Yaskawa INFORM job: u_tourne2TRJ4.JBI

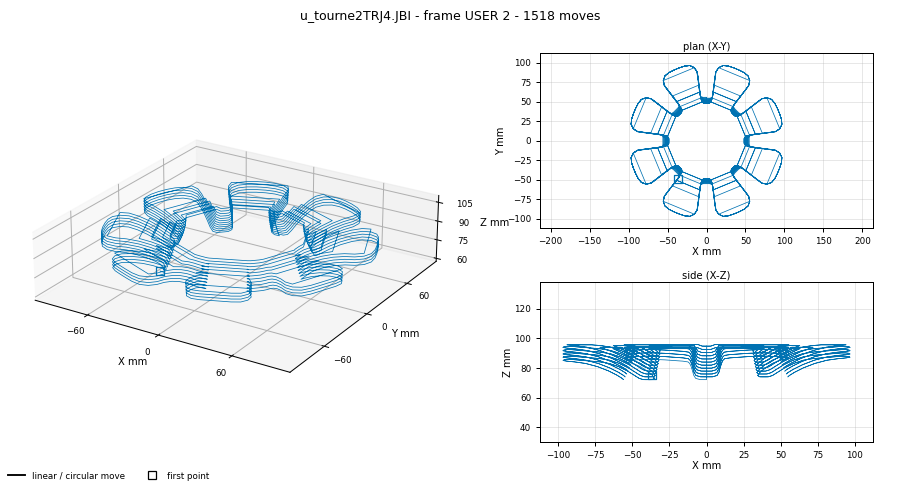
[picture p0: tool path of u_tourne2TRJ4.JBI in frame USER 2, 1518 of 1518 moves have a stored position in this frame; points joined in program order, loops and branches not executed]
/JOB
//NAME u_tourne2TRJ4
///FOLDERNAME DEMO
//POS
///NPOS 1518,0,0,0,0,0
///USER 2
///TOOL 7
///POSTYPE USER
///RECTAN
///RCONF 1,0,0,0,0,0,0,0,0,0,0,0,0,0,0,0,0,0,0,0,0,0,0,0
C00000=-36.517,-48.718,75.143,178.8248,-1.7081,0.0000
C00001=-35.037,-45.351,73.015,-179.8799,17.3496,0.0000
C00002=-36.538,-42.505,72.166,160.0584,24.5518,0.0000
C00003=-38.303,-40.803,72.129,156.0394,22.3811,0.0000
C00004=-39.567,-39.567,72.154,156.8184,23.1816,0.0000
C00005=-40.803,-38.303,72.129,157.6189,23.9606,0.0000
C00006=-42.506,-36.538,72.166,155.4482,19.9416,0.0000
C00007=-45.352,-35.037,73.015,162.6504,-0.1201,0.0000
C00008=-48.718,-36.517,75.143,-178.2919,1.1752,0.0000
C00009=-53.324,-40.007,78.036,-176.9022,2.2727,0.0000
C00010=-59.196,-44.618,80.927,-176.4763,2.6299,0.0000
C00011=-65.578,-49.604,83.062,-176.2458,2.8088,0.0000
C00012=-71.524,-53.949,84.088,-176.0063,2.0395,0.0000
C00013=-77.795,-55.184,84.621,-177.1914,-0.2581,0.0000
C00014=-83.601,-53.037,85.050,-178.9055,-0.7851,0.0000
C00015=-87.741,-47.957,85.481,-179.9599,-0.0745,0.0000
C00016=-90.934,-41.602,85.762,-179.9943,-0.0115,0.0000
C00017=-93.717,-34.883,85.762,-179.9943,-0.0115,0.0000
C00018=-95.953,-28.131,85.481,-179.9771,-0.0859,0.0000
C00019=-96.617,-21.612,85.050,179.7822,-1.3294,0.0000
C00020=-94.030,-15.989,84.621,178.1936,-2.1673,0.0000
C00021=-88.723,-12.427,84.088,175.7376,-1.3849,0.0000
C00022=-81.446,-11.295,83.062,175.3653,-0.6668,0.0000
C00023=-73.408,-10.308,80.927,175.6470,-0.6321,0.0000
C00024=-65.995,-9.417,78.036,176.2042,-0.5857,0.0000
C00025=-60.270,-8.627,75.143,177.9597,-0.3784,0.0000
C00026=-56.844,-7.293,73.015,-167.4661,12.3794,0.0000
C00027=-55.892,-4.219,72.166,-176.1983,30.0937,0.0000
C00028=-55.936,-1.768,72.129,178.6805,31.1908,0.0000
C00029=-55.957,0.000,72.154,180.0000,31.1976,0.0000
C00030=-55.936,1.767,72.129,-178.6805,31.1908,0.0000
C00031=-55.892,4.220,72.166,176.1916,30.0937,0.0000
C00032=-56.844,7.293,73.015,167.4661,12.3794,0.0000
C00033=-60.270,8.627,75.143,-177.9597,-0.3784,0.0000
C00034=-65.995,9.417,78.036,-176.2042,-0.5857,0.0000
C00035=-73.408,10.308,80.927,-175.6470,-0.6321,0.0000
C00036=-81.446,11.295,83.062,-175.3653,-0.6668,0.0000
C00037=-88.723,12.427,84.088,-175.7376,-1.3849,0.0000
C00038=-94.030,15.989,84.621,-178.1936,-2.1673,0.0000
C00039=-96.617,21.612,85.050,-179.7822,-1.3294,0.0000
C00040=-95.953,28.131,85.481,179.9771,-0.0859,0.0000
C00041=-93.717,34.883,85.762,179.9943,-0.0115,0.0000
C00042=-90.934,41.602,85.762,179.9943,-0.0115,0.0000
C00043=-87.741,47.957,85.481,179.9599,-0.0745,0.0000
C00044=-83.601,53.037,85.050,178.9055,-0.7851,0.0000
C00045=-77.795,55.184,84.621,177.1914,-0.2581,0.0000
C00046=-71.524,53.949,84.088,176.0063,2.0395,0.0000
C00047=-65.578,49.604,83.062,176.2458,2.8088,0.0000
C00048=-59.196,44.618,80.927,176.4763,2.6299,0.0000
C00049=-53.324,40.007,78.036,176.9022,2.2727,0.0000
C00050=-48.718,36.517,75.143,178.2919,1.1752,0.0000
C00051=-45.351,35.037,73.015,-162.6504,-0.1201,0.0000
C00052=-42.505,36.538,72.166,-155.4482,19.9416,0.0000
C00053=-40.803,38.303,72.129,-157.6189,23.9606,0.0000
C00054=-39.567,39.567,72.154,-156.8184,23.1816,0.0000
C00055=-38.303,40.803,72.129,-156.0394,22.3811,0.0000
C00056=-36.538,42.506,72.166,-160.0584,24.5518,0.0000
C00057=-35.037,45.352,73.015,179.8799,17.3496,0.0000
C00058=-36.517,48.718,75.143,-178.8248,-1.7081,0.0000
C00059=-40.007,53.324,78.036,-177.7273,-3.0978,0.0000
C00060=-44.618,59.196,80.927,-177.3701,-3.5237,0.0000
C00061=-49.604,65.578,83.062,-177.1912,-3.7542,0.0000
C00062=-53.949,71.524,84.088,-177.9605,-3.9937,0.0000
C00063=-55.184,77.795,84.621,179.7419,-2.8086,0.0000
C00064=-53.037,83.601,85.050,179.2149,-1.0945,0.0000
C00065=-47.957,87.741,85.481,179.9255,-0.0401,0.0000
C00066=-41.602,90.934,85.762,179.9885,-0.0057,0.0000
C00067=-34.883,93.717,85.762,179.9885,-0.0057,0.0000
C00068=-28.131,95.953,85.481,179.9141,-0.0229,0.0000
C00069=-21.612,96.617,85.050,178.6706,0.2178,0.0000
C00070=-15.989,94.030,84.621,177.8327,1.8064,0.0000
C00071=-12.427,88.723,84.088,178.6151,4.2624,0.0000
C00072=-11.295,81.446,83.062,179.3332,4.6347,0.0000
C00073=-10.308,73.408,80.927,179.3679,4.3530,0.0000
C00074=-9.417,65.995,78.036,179.4143,3.7958,0.0000
C00075=-8.627,60.270,75.143,179.6216,2.0403,0.0000
C00076=-7.293,56.844,73.015,-167.6206,-12.5339,0.0000
C00077=-4.220,55.892,72.166,-149.9063,-3.8084,0.0000
C00078=-1.767,55.936,72.129,-148.8092,1.3195,0.0000
C00079=0.000,55.957,72.154,-148.8024,-0.0000,0.0000
C00080=0.000,54.840,74.049,-150.2587,-0.0000,0.0000
C00081=1.666,54.823,74.024,-150.2658,-1.1877,0.0000
C00082=4.048,54.790,74.062,-151.4221,3.8700,0.0000
C00083=7.088,55.804,74.943,-168.9171,11.6612,0.0000
C00084=8.393,59.388,77.145,179.6273,-2.1319,0.0000
C00085=9.180,65.335,80.122,179.4719,-3.5317,0.0000
C00086=10.089,72.980,83.074,179.4487,-3.8705,0.0000
C00087=11.094,81.206,85.240,179.4429,-3.9856,0.0000
C00088=12.226,88.613,86.276,178.8517,-3.5956,0.0000
C00089=15.808,94.009,86.813,178.2001,-1.5192,0.0000
C00090=21.475,96.642,87.246,178.8998,-0.1834,0.0000
C00091=28.048,95.980,87.679,179.9312,0.0229,0.0000
C00092=34.856,93.728,87.962,179.9943,0.0057,0.0000
C00093=41.629,90.922,87.962,179.9943,0.0057,0.0000
C00094=48.035,87.701,87.679,179.9370,0.0344,0.0000
C00095=53.151,83.521,87.246,179.3525,0.9054,0.0000
C00096=55.296,77.652,86.813,179.7993,2.3440,0.0000
C00097=54.014,71.304,86.276,-178.2664,3.3554,0.0000
C00098=49.577,65.266,85.240,-177.5775,3.2132,0.0000
C00099=44.470,58.738,83.074,-177.6468,3.1267,0.0000
C00100=39.708,52.690,80.122,-177.8713,2.8736,0.0000
C00101=36.059,47.928,77.145,-178.7560,1.7711,0.0000
C00102=34.447,44.472,74.943,179.5711,-15.8793,0.0000
C00103=35.880,41.605,74.062,-161.3594,-23.4144,0.0000
C00104=37.588,39.944,74.024,-157.2874,-21.2658,0.0000
C00105=38.778,38.778,74.049,-158.0009,-21.9991,0.0000
C00106=39.943,37.588,74.024,-158.7342,-22.7126,0.0000
C00107=41.605,35.880,74.062,-156.5880,-18.6327,0.0000
C00108=44.472,34.447,74.943,-164.1207,0.4289,0.0000
C00109=47.928,36.059,77.145,178.2289,-1.2440,0.0000
C00110=52.690,39.708,80.122,177.1264,-2.1287,0.0000
C00111=58.738,44.470,83.074,176.8733,-2.3532,0.0000
C00112=65.266,49.577,85.240,176.7868,-2.4225,0.0000
C00113=71.304,54.014,86.276,176.6446,-1.7336,0.0000
C00114=77.652,55.296,86.813,177.6560,0.2007,0.0000
C00115=83.521,53.151,87.246,179.0946,0.6475,0.0000
C00116=87.701,48.035,87.679,179.9656,0.0630,0.0000
C00117=90.922,41.629,87.962,179.9943,0.0057,0.0000
C00118=93.728,34.856,87.962,179.9943,0.0057,0.0000
C00119=95.980,28.048,87.679,179.9771,0.0688,0.0000
C00120=96.642,21.475,87.246,-179.8166,1.1002,0.0000
C00121=94.009,15.808,86.813,-178.4808,1.7999,0.0000
C00122=88.613,12.226,86.276,-176.4044,1.1483,0.0000
C00123=81.206,11.094,85.240,-176.0144,0.5571,0.0000
C00124=72.980,10.089,83.074,-176.1295,0.5513,0.0000
C00125=65.335,9.180,80.122,-176.4683,0.5281,0.0000
C00126=59.388,8.393,77.145,-177.8681,0.3727,0.0000
C00127=55.804,7.088,74.943,168.3388,-11.0829,0.0000
C00128=54.790,4.048,74.062,176.1300,-28.5779,0.0000
C00129=54.823,1.666,74.024,-178.8123,-29.7342,0.0000
C00130=54.840,0.000,74.049,-180.0000,-29.7413,0.0000
C00131=54.823,-1.665,74.024,178.8123,-29.7342,0.0000
C00132=54.790,-4.048,74.062,-176.1304,-28.5752,0.0000
C00133=55.804,-7.088,74.943,-168.3388,-11.0829,0.0000
C00134=59.388,-8.393,77.145,177.8681,0.3727,0.0000
C00135=65.335,-9.180,80.122,176.4683,0.5281,0.0000
C00136=72.980,-10.089,83.074,176.1295,0.5513,0.0000
C00137=81.206,-11.094,85.240,176.0144,0.5571,0.0000
C00138=88.613,-12.226,86.276,176.4044,1.1483,0.0000
C00139=94.009,-15.808,86.813,178.4808,1.7999,0.0000
C00140=96.642,-21.475,87.246,179.8166,1.1002,0.0000
C00141=95.980,-28.048,87.679,-179.9771,0.0688,0.0000
C00142=93.728,-34.856,87.962,-179.9943,0.0057,0.0000
C00143=90.922,-41.629,87.962,-179.9943,0.0057,0.0000
C00144=87.701,-48.035,87.679,-179.9656,0.0630,0.0000
C00145=83.521,-53.151,87.246,-179.0946,0.6475,0.0000
C00146=77.652,-55.296,86.813,-177.6560,0.2007,0.0000
C00147=71.304,-54.014,86.276,-176.6446,-1.7336,0.0000
C00148=65.266,-49.577,85.240,-176.7868,-2.4225,0.0000
C00149=58.738,-44.470,83.074,-176.8733,-2.3532,0.0000
C00150=52.690,-39.708,80.122,-177.1264,-2.1287,0.0000
C00151=47.928,-36.059,77.145,-178.2289,-1.2440,0.0000
C00152=44.472,-34.447,74.943,164.1207,0.4289,0.0000
C00153=41.605,-35.880,74.062,156.5856,-18.6406,0.0000
C00154=39.944,-37.588,74.024,158.7342,-22.7126,0.0000
C00155=38.778,-38.778,74.049,158.0009,-21.9991,0.0000
C00156=37.588,-39.943,74.024,157.2874,-21.2658,0.0000
C00157=35.880,-41.605,74.062,161.3673,-23.4120,0.0000
C00158=34.447,-44.472,74.943,-179.5711,-15.8793,0.0000
C00159=36.059,-47.928,77.145,178.7560,1.7711,0.0000
C00160=39.708,-52.690,80.122,177.8713,2.8736,0.0000
C00161=44.470,-58.738,83.074,177.6468,3.1267,0.0000
C00162=49.577,-65.266,85.240,177.5775,3.2132,0.0000
C00163=54.014,-71.304,86.276,178.2664,3.3554,0.0000
C00164=55.296,-77.652,86.813,-179.7993,2.3440,0.0000
C00165=53.151,-83.521,87.246,-179.3525,0.9054,0.0000
C00166=48.035,-87.701,87.679,-179.9370,0.0344,0.0000
C00167=41.629,-90.922,87.962,-179.9943,0.0057,0.0000
C00168=34.856,-93.728,87.962,-179.9943,0.0057,0.0000
C00169=28.048,-95.980,87.679,-179.9312,0.0229,0.0000
C00170=21.475,-96.642,87.246,-178.8998,-0.1834,0.0000
C00171=15.808,-94.009,86.813,-178.2001,-1.5192,0.0000
C00172=12.226,-88.613,86.276,-178.8517,-3.5956,0.0000
C00173=11.094,-81.206,85.240,-179.4429,-3.9856,0.0000
C00174=10.089,-72.980,83.074,-179.4487,-3.8705,0.0000
C00175=9.180,-65.335,80.122,-179.4719,-3.5317,0.0000
C00176=8.393,-59.388,77.145,-179.6273,-2.1319,0.0000
C00177=7.088,-55.804,74.943,168.9171,11.6612,0.0000
C00178=4.048,-54.790,74.062,151.4221,3.8700,0.0000
C00179=1.666,-54.823,74.024,150.2658,-1.1877,0.0000
C00180=0.000,-54.840,74.049,150.2587,-0.0000,0.0000
C00181=0.000,-54.840,74.049,150.2587,-0.0000,0.0000
C00182=-1.665,-54.823,74.024,150.2658,1.1877,0.0000
C00183=-4.048,-54.790,74.062,151.4248,-3.8696,0.0000
C00184=-7.088,-55.804,74.943,168.9171,-11.6612,0.0000
C00185=-8.393,-59.388,77.145,-179.6273,2.1319,0.0000
C00186=-9.180,-65.335,80.122,-179.4719,3.5317,0.0000
C00187=-10.089,-72.980,83.074,-179.4487,3.8705,0.0000
C00188=-11.094,-81.206,85.240,-179.4429,3.9856,0.0000
C00189=-12.226,-88.613,86.276,-178.8517,3.5956,0.0000
C00190=-15.808,-94.009,86.813,-178.2001,1.5192,0.0000
C00191=-21.475,-96.642,87.246,-178.8998,0.1834,0.0000
C00192=-28.048,-95.980,87.679,-179.9312,-0.0229,0.0000
C00193=-34.856,-93.728,87.962,-179.9943,-0.0057,0.0000
C00194=-41.629,-90.922,87.962,-179.9943,-0.0057,0.0000
C00195=-48.035,-87.701,87.679,-179.9370,-0.0344,0.0000
C00196=-53.151,-83.521,87.246,-179.3525,-0.9054,0.0000
C00197=-55.296,-77.652,86.813,-179.7993,-2.3440,0.0000
C00198=-54.014,-71.304,86.276,178.2664,-3.3554,0.0000
C00199=-49.577,-65.266,85.240,177.5775,-3.2132,0.0000
C00200=-44.470,-58.738,83.074,177.6468,-3.1267,0.0000
C00201=-39.708,-52.690,80.122,177.8713,-2.8736,0.0000
C00202=-36.059,-47.928,77.145,178.7560,-1.7711,0.0000
C00203=-34.447,-44.472,74.943,-179.5711,15.8793,0.0000
C00204=-35.880,-41.605,74.062,161.3594,23.4144,0.0000
C00205=-37.588,-39.944,74.024,157.2874,21.2658,0.0000
C00206=-38.778,-38.778,74.049,158.0009,21.9991,0.0000
C00207=-39.943,-37.588,74.024,158.7342,22.7126,0.0000
C00208=-41.605,-35.880,74.062,156.5880,18.6327,0.0000
C00209=-44.472,-34.447,74.943,164.1207,-0.4289,0.0000
C00210=-47.928,-36.059,77.145,-178.2289,1.2440,0.0000
C00211=-52.690,-39.708,80.122,-177.1264,2.1287,0.0000
C00212=-58.738,-44.470,83.074,-176.8733,2.3532,0.0000
C00213=-65.266,-49.577,85.240,-176.7868,2.4225,0.0000
C00214=-71.304,-54.014,86.276,-176.6446,1.7336,0.0000
C00215=-77.652,-55.296,86.813,-177.6560,-0.2007,0.0000
C00216=-83.521,-53.151,87.246,-179.0946,-0.6475,0.0000
C00217=-87.701,-48.035,87.679,-179.9656,-0.0630,0.0000
C00218=-90.922,-41.629,87.962,-179.9943,-0.0057,0.0000
C00219=-93.728,-34.856,87.962,-179.9943,-0.0057,0.0000
C00220=-95.980,-28.048,87.679,-179.9771,-0.0688,0.0000
C00221=-96.642,-21.475,87.246,179.8166,-1.1002,0.0000
C00222=-94.009,-15.808,86.813,178.4808,-1.7999,0.0000
C00223=-88.613,-12.226,86.276,176.4044,-1.1483,0.0000
C00224=-81.206,-11.094,85.240,176.0144,-0.5571,0.0000
C00225=-72.980,-10.089,83.074,176.1295,-0.5513,0.0000
C00226=-65.335,-9.180,80.122,176.4683,-0.5281,0.0000
C00227=-59.388,-8.393,77.145,177.8681,-0.3727,0.0000
C00228=-55.804,-7.088,74.943,-168.3388,11.0829,0.0000
C00229=-54.790,-4.048,74.062,-176.1300,28.5779,0.0000
C00230=-54.823,-1.666,74.024,178.8123,29.7342,0.0000
C00231=-54.840,0.000,74.049,180.0000,29.7413,0.0000
C00232=-54.823,1.665,74.024,-178.8123,29.7342,0.0000
C00233=-54.790,4.048,74.062,176.1304,28.5752,0.0000
C00234=-55.804,7.088,74.943,168.3388,11.0829,0.0000
C00235=-59.388,8.393,77.145,-177.8681,-0.3727,0.0000
C00236=-65.335,9.180,80.122,-176.4683,-0.5281,0.0000
C00237=-72.980,10.089,83.074,-176.1295,-0.5513,0.0000
C00238=-81.206,11.094,85.240,-176.0144,-0.5571,0.0000
C00239=-88.613,12.226,86.276,-176.4044,-1.1483,0.0000
C00240=-94.009,15.808,86.813,-178.4808,-1.7999,0.0000
C00241=-96.642,21.475,87.246,-179.8166,-1.1002,0.0000
C00242=-95.980,28.048,87.679,179.9771,-0.0688,0.0000
C00243=-93.728,34.856,87.962,179.9943,-0.0057,0.0000
C00244=-90.922,41.629,87.962,179.9943,-0.0057,0.0000
C00245=-87.701,48.035,87.679,179.9656,-0.0630,0.0000
C00246=-83.521,53.151,87.246,179.0946,-0.6475,0.0000
C00247=-77.652,55.296,86.813,177.6560,-0.2007,0.0000
C00248=-71.304,54.014,86.276,176.6446,1.7336,0.0000
C00249=-65.266,49.577,85.240,176.7868,2.4225,0.0000
C00250=-58.738,44.470,83.074,176.8733,2.3532,0.0000
C00251=-52.690,39.708,80.122,177.1264,2.1287,0.0000
C00252=-47.928,36.059,77.145,178.2289,1.2440,0.0000
C00253=-44.472,34.447,74.943,-164.1207,-0.4289,0.0000
C00254=-41.605,35.880,74.062,-156.5856,18.6406,0.0000
C00255=-39.944,37.588,74.024,-158.7342,22.7126,0.0000
C00256=-38.778,38.778,74.049,-158.0009,21.9991,0.0000
C00257=-37.588,39.943,74.024,-157.2874,21.2658,0.0000
C00258=-35.880,41.605,74.062,-161.3673,23.4120,0.0000
C00259=-34.447,44.472,74.943,179.5711,15.8793,0.0000
C00260=-36.059,47.928,77.145,-178.7560,-1.7711,0.0000
C00261=-39.708,52.690,80.122,-177.8713,-2.8736,0.0000
C00262=-44.470,58.738,83.074,-177.6468,-3.1267,0.0000
C00263=-49.577,65.266,85.240,-177.5775,-3.2132,0.0000
C00264=-54.014,71.304,86.276,-178.2664,-3.3554,0.0000
C00265=-55.296,77.652,86.813,179.7993,-2.3440,0.0000
C00266=-53.151,83.521,87.246,179.3525,-0.9054,0.0000
C00267=-48.035,87.701,87.679,179.9370,-0.0344,0.0000
C00268=-41.629,90.922,87.962,179.9943,-0.0057,0.0000
C00269=-34.856,93.728,87.962,179.9943,-0.0057,0.0000
C00270=-28.048,95.980,87.679,179.9312,-0.0229,0.0000
C00271=-21.475,96.642,87.246,178.8998,0.1834,0.0000
C00272=-15.808,94.009,86.813,178.2001,1.5192,0.0000
C00273=-12.226,88.613,86.276,178.8517,3.5956,0.0000
C00274=-11.094,81.206,85.240,179.4429,3.9856,0.0000
C00275=-10.089,72.980,83.074,179.4487,3.8705,0.0000
C00276=-9.180,65.335,80.122,179.4719,3.5317,0.0000
C00277=-8.393,59.388,77.145,179.6273,2.1319,0.0000
C00278=-7.088,55.804,74.943,-168.9171,-11.6612,0.0000
C00279=-4.048,54.790,74.062,-151.4248,-3.8696,0.0000
C00280=-1.665,54.823,74.024,-150.2658,1.1877,0.0000
C00281=0.000,54.840,74.049,-150.2587,-0.0000,0.0000
C00282=0.000,53.776,75.975,-151.8999,-0.0000,0.0000
C00283=1.568,53.762,75.948,-151.9022,-1.0587,0.0000
C00284=3.884,53.739,75.988,-153.1141,3.8747,0.0000
C00285=6.894,54.818,76.900,-170.1659,10.7275,0.0000
C00286=8.175,58.565,79.173,179.6445,-2.1491,0.0000
C00287=8.965,64.737,82.228,179.5352,-3.2161,0.0000
C00288=9.898,72.606,85.234,179.5351,-3.3365,0.0000
C00289=10.924,81.005,87.424,179.5523,-3.2736,0.0000
C00290=12.061,88.524,88.468,179.0993,-2.8721,0.0000
C00291=15.662,93.991,89.008,178.5901,-1.1979,0.0000
C00292=21.365,96.662,89.443,179.1520,-0.1433,0.0000
C00293=27.983,96.002,89.878,179.9484,0.0172,0.0000
C00294=34.834,93.736,90.162,179.9943,0.0000,0.0000
C00295=41.650,90.913,90.162,179.9943,0.0000,0.0000
C00296=48.097,87.670,89.878,179.9542,0.0286,0.0000
C00297=53.243,83.458,89.443,179.5015,0.7048,0.0000
C00298=55.387,77.537,89.008,179.8510,1.8452,0.0000
C00299=54.067,71.124,88.468,-178.6060,2.6718,0.0000
C00300=49.554,65.004,87.424,-178.0035,2.6325,0.0000
C00301=44.341,58.339,85.234,-177.9691,2.6898,0.0000
C00302=39.437,52.115,82.228,-178.0553,2.6036,0.0000
C00303=35.631,47.192,79.173,-178.7331,1.7711,0.0000
C00304=33.888,43.637,76.900,179.3493,-14.3892,0.0000
C00305=35.253,40.746,75.988,-162.7468,-22.1158,0.0000
C00306=36.906,39.124,75.948,-158.6649,-20.0217,0.0000
C00307=38.025,38.025,75.975,-159.3181,-20.6819,0.0000
C00308=39.124,36.906,75.948,-159.9783,-21.3351,0.0000
C00309=40.746,35.253,75.988,-157.8842,-17.2532,0.0000
C00310=43.637,33.888,76.901,-165.6108,0.6507,0.0000
C00311=47.192,35.631,79.173,178.2289,-1.2669,0.0000
C00312=52.115,39.437,82.228,177.3964,-1.9447,0.0000
C00313=58.339,44.341,85.234,177.3102,-2.0309,0.0000
C00314=65.004,49.554,87.424,177.3675,-1.9965,0.0000
C00315=71.124,54.067,88.468,177.3282,-1.3940,0.0000
C00316=77.537,55.387,89.008,178.1548,0.1490,0.0000
C00317=83.458,53.243,89.443,179.2952,0.4985,0.0000
C00318=87.670,48.097,89.878,179.9714,0.0458,0.0000
C00319=90.913,41.650,90.162,180.0000,0.0057,0.0000
C00320=93.736,34.834,90.162,180.0000,0.0057,0.0000
C00321=96.002,27.983,89.878,179.9828,0.0516,0.0000
C00322=96.662,21.365,89.443,-179.8567,0.8480,0.0000
C00323=93.991,15.662,89.008,-178.8021,1.4099,0.0000
C00324=88.524,12.061,88.468,-177.1279,0.9007,0.0000
C00325=81.005,10.924,87.424,-176.7264,0.4477,0.0000
C00326=72.606,9.898,85.234,-176.6635,0.4649,0.0000
C00327=64.737,8.965,82.228,-176.7839,0.4648,0.0000
C00328=58.565,8.175,79.173,-177.8509,0.3555,0.0000
C00329=54.818,6.894,76.900,169.2725,-9.8341,0.0000
C00330=53.739,3.884,75.988,176.1253,-26.8859,0.0000
C00331=53.762,1.568,75.948,-178.9413,-28.0978,0.0000
C00332=53.776,0.000,75.975,-180.0000,-28.1001,0.0000
C00333=53.762,-1.568,75.948,178.9413,-28.0978,0.0000
C00334=53.739,-3.885,75.988,-176.1253,-26.8859,0.0000
C00335=54.819,-6.894,76.901,-169.2725,-9.8341,0.0000
C00336=58.565,-8.175,79.173,177.8509,0.3555,0.0000
C00337=64.737,-8.965,82.228,176.7839,0.4648,0.0000
C00338=72.606,-9.898,85.234,176.6635,0.4649,0.0000
C00339=81.005,-10.924,87.424,176.7264,0.4477,0.0000
C00340=88.524,-12.061,88.468,177.1279,0.9007,0.0000
C00341=93.991,-15.662,89.008,178.8021,1.4099,0.0000
C00342=96.662,-21.365,89.443,179.8567,0.8480,0.0000
C00343=96.002,-27.983,89.878,-179.9828,0.0516,0.0000
C00344=93.736,-34.834,90.162,-180.0000,0.0057,0.0000
C00345=90.913,-41.650,90.162,-180.0000,0.0057,0.0000
C00346=87.670,-48.097,89.878,-179.9714,0.0458,0.0000
C00347=83.458,-53.243,89.443,-179.2952,0.4985,0.0000
C00348=77.537,-55.387,89.008,-178.1548,0.1490,0.0000
C00349=71.124,-54.067,88.468,-177.3282,-1.3940,0.0000
C00350=65.004,-49.554,87.424,-177.3675,-1.9965,0.0000
C00351=58.339,-44.341,85.234,-177.3102,-2.0309,0.0000
C00352=52.115,-39.437,82.228,-177.3964,-1.9447,0.0000
C00353=47.192,-35.631,79.173,-178.2289,-1.2669,0.0000
C00354=43.637,-33.888,76.900,165.6108,0.6507,0.0000
C00355=40.746,-35.253,75.988,157.8842,-17.2532,0.0000
C00356=39.124,-36.906,75.948,159.9783,-21.3351,0.0000
C00357=38.025,-38.025,75.975,159.3181,-20.6819,0.0000
C00358=36.906,-39.124,75.948,158.6649,-20.0217,0.0000
C00359=35.253,-40.746,75.988,162.7468,-22.1158,0.0000
C00360=33.888,-43.637,76.901,-179.3493,-14.3892,0.0000
C00361=35.631,-47.192,79.173,178.7331,1.7711,0.0000
C00362=39.437,-52.115,82.228,178.0553,2.6036,0.0000
C00363=44.341,-58.339,85.234,177.9691,2.6898,0.0000
C00364=49.554,-65.004,87.424,178.0035,2.6325,0.0000
C00365=54.067,-71.124,88.468,178.6060,2.6718,0.0000
C00366=55.387,-77.537,89.008,-179.8510,1.8452,0.0000
C00367=53.243,-83.458,89.443,-179.5015,0.7048,0.0000
C00368=48.097,-87.670,89.878,-179.9542,0.0286,0.0000
C00369=41.650,-90.913,90.162,-179.9943,0.0000,0.0000
C00370=34.834,-93.736,90.162,-179.9943,0.0000,0.0000
C00371=27.983,-96.002,89.878,-179.9484,0.0172,0.0000
C00372=21.365,-96.662,89.443,-179.1520,-0.1433,0.0000
C00373=15.662,-93.991,89.008,-178.5901,-1.1979,0.0000
C00374=12.061,-88.524,88.468,-179.0993,-2.8721,0.0000
C00375=10.924,-81.005,87.424,-179.5523,-3.2736,0.0000
C00376=9.898,-72.606,85.234,-179.5351,-3.3365,0.0000
C00377=8.965,-64.737,82.228,-179.5352,-3.2161,0.0000
C00378=8.175,-58.565,79.173,-179.6445,-2.1491,0.0000
C00379=6.894,-54.818,76.900,170.1659,10.7275,0.0000
C00380=3.884,-53.739,75.988,153.1141,3.8747,0.0000
C00381=1.568,-53.762,75.948,151.9022,-1.0587,0.0000
C00382=0.000,-53.776,75.975,151.8999,-0.0000,0.0000
C00383=0.000,-53.776,75.975,151.8999,-0.0000,0.0000
C00384=-1.568,-53.762,75.948,151.9022,1.0587,0.0000
C00385=-3.885,-53.739,75.988,153.1141,-3.8747,0.0000
C00386=-6.894,-54.819,76.901,170.1659,-10.7275,0.0000
C00387=-8.175,-58.565,79.173,-179.6445,2.1491,0.0000
C00388=-8.965,-64.737,82.228,-179.5352,3.2161,0.0000
C00389=-9.898,-72.606,85.234,-179.5351,3.3365,0.0000
C00390=-10.924,-81.005,87.424,-179.5523,3.2736,0.0000
C00391=-12.061,-88.524,88.468,-179.0993,2.8721,0.0000
C00392=-15.662,-93.991,89.008,-178.5901,1.1979,0.0000
C00393=-21.365,-96.662,89.443,-179.1520,0.1433,0.0000
C00394=-27.983,-96.002,89.878,-179.9484,-0.0172,0.0000
C00395=-34.834,-93.736,90.162,-179.9943,-0.0000,0.0000
C00396=-41.650,-90.913,90.162,-179.9943,-0.0000,0.0000
C00397=-48.097,-87.670,89.878,-179.9542,-0.0286,0.0000
C00398=-53.243,-83.458,89.443,-179.5015,-0.7048,0.0000
C00399=-55.387,-77.537,89.008,-179.8510,-1.8452,0.0000
C00400=-54.067,-71.124,88.468,178.6060,-2.6718,0.0000
C00401=-49.554,-65.004,87.424,178.0035,-2.6325,0.0000
C00402=-44.341,-58.339,85.234,177.9691,-2.6898,0.0000
C00403=-39.437,-52.115,82.228,178.0553,-2.6036,0.0000
C00404=-35.631,-47.192,79.173,178.7331,-1.7711,0.0000
C00405=-33.888,-43.637,76.900,-179.3493,14.3892,0.0000
C00406=-35.253,-40.746,75.988,162.7468,22.1158,0.0000
C00407=-36.906,-39.124,75.948,158.6649,20.0217,0.0000
C00408=-38.025,-38.025,75.975,159.3181,20.6819,0.0000
C00409=-39.124,-36.906,75.948,159.9783,21.3351,0.0000
C00410=-40.746,-35.253,75.988,157.8842,17.2532,0.0000
C00411=-43.637,-33.888,76.901,165.6108,-0.6507,0.0000
C00412=-47.192,-35.631,79.173,-178.2289,1.2669,0.0000
C00413=-52.115,-39.437,82.228,-177.3964,1.9447,0.0000
C00414=-58.339,-44.341,85.234,-177.3102,2.0309,0.0000
C00415=-65.004,-49.554,87.424,-177.3675,1.9965,0.0000
C00416=-71.124,-54.067,88.468,-177.3282,1.3940,0.0000
C00417=-77.537,-55.387,89.008,-178.1548,-0.1490,0.0000
C00418=-83.458,-53.243,89.443,-179.2952,-0.4985,0.0000
C00419=-87.670,-48.097,89.878,-179.9714,-0.0458,0.0000
C00420=-90.913,-41.650,90.162,-180.0000,-0.0057,0.0000
C00421=-93.736,-34.834,90.162,-180.0000,-0.0057,0.0000
C00422=-96.002,-27.983,89.878,-179.9828,-0.0516,0.0000
C00423=-96.662,-21.365,89.443,179.8567,-0.8480,0.0000
C00424=-93.991,-15.662,89.008,178.8021,-1.4099,0.0000
C00425=-88.524,-12.061,88.468,177.1279,-0.9007,0.0000
C00426=-81.005,-10.924,87.424,176.7264,-0.4477,0.0000
C00427=-72.606,-9.898,85.234,176.6635,-0.4649,0.0000
C00428=-64.737,-8.965,82.228,176.7839,-0.4648,0.0000
C00429=-58.565,-8.175,79.173,177.8509,-0.3555,0.0000
C00430=-54.818,-6.894,76.900,-169.2725,9.8341,0.0000
C00431=-53.739,-3.884,75.988,-176.1253,26.8859,0.0000
C00432=-53.762,-1.568,75.948,178.9413,28.0978,0.0000
C00433=-53.776,0.000,75.975,180.0000,28.1001,0.0000
C00434=-53.762,1.568,75.948,-178.9413,28.0978,0.0000
C00435=-53.739,3.885,75.988,176.1253,26.8859,0.0000
C00436=-54.819,6.894,76.901,169.2725,9.8341,0.0000
C00437=-58.565,8.175,79.173,-177.8509,-0.3555,0.0000
C00438=-64.737,8.965,82.228,-176.7839,-0.4648,0.0000
C00439=-72.606,9.898,85.234,-176.6635,-0.4649,0.0000
C00440=-81.005,10.924,87.424,-176.7264,-0.4477,0.0000
C00441=-88.524,12.061,88.468,-177.1279,-0.9007,0.0000
C00442=-93.991,15.662,89.008,-178.8021,-1.4099,0.0000
C00443=-96.662,21.365,89.443,-179.8567,-0.8480,0.0000
C00444=-96.002,27.983,89.878,179.9828,-0.0516,0.0000
C00445=-93.736,34.834,90.162,180.0000,-0.0057,0.0000
C00446=-90.913,41.650,90.162,180.0000,-0.0057,0.0000
C00447=-87.670,48.097,89.878,179.9714,-0.0458,0.0000
C00448=-83.458,53.243,89.443,179.2952,-0.4985,0.0000
C00449=-77.537,55.387,89.008,178.1548,-0.1490,0.0000
C00450=-71.124,54.067,88.468,177.3282,1.3940,0.0000
C00451=-65.004,49.554,87.424,177.3675,1.9965,0.0000
C00452=-58.339,44.341,85.234,177.3102,2.0309,0.0000
C00453=-52.115,39.437,82.228,177.3964,1.9447,0.0000
C00454=-47.192,35.631,79.173,178.2289,1.2669,0.0000
C00455=-43.637,33.888,76.900,-165.6108,-0.6507,0.0000
C00456=-40.746,35.253,75.988,-157.8842,17.2532,0.0000
C00457=-39.124,36.906,75.948,-159.9783,21.3351,0.0000
C00458=-38.025,38.025,75.975,-159.3181,20.6819,0.0000
C00459=-36.906,39.124,75.948,-158.6649,20.0217,0.0000
C00460=-35.253,40.746,75.988,-162.7468,22.1158,0.0000
C00461=-33.888,43.637,76.901,179.3493,14.3892,0.0000
C00462=-35.631,47.192,79.173,-178.7331,-1.7711,0.0000
C00463=-39.437,52.115,82.228,-178.0553,-2.6036,0.0000
C00464=-44.341,58.339,85.234,-177.9691,-2.6898,0.0000
C00465=-49.554,65.004,87.424,-178.0035,-2.6325,0.0000
C00466=-54.067,71.124,88.468,-178.6060,-2.6718,0.0000
C00467=-55.387,77.537,89.008,179.8510,-1.8452,0.0000
C00468=-53.243,83.458,89.443,179.5015,-0.7048,0.0000
C00469=-48.097,87.670,89.878,179.9542,-0.0286,0.0000
C00470=-41.650,90.913,90.162,179.9943,-0.0000,0.0000
C00471=-34.834,93.736,90.162,179.9943,-0.0000,0.0000
C00472=-27.983,96.002,89.878,179.9484,-0.0172,0.0000
C00473=-21.365,96.662,89.443,179.1520,0.1433,0.0000
C00474=-15.662,93.991,89.008,178.5901,1.1979,0.0000
C00475=-12.061,88.524,88.468,179.0993,2.8721,0.0000
C00476=-10.924,81.005,87.424,179.5523,3.2736,0.0000
C00477=-9.898,72.606,85.234,179.5351,3.3365,0.0000
C00478=-8.965,64.737,82.228,179.5352,3.2161,0.0000
C00479=-8.175,58.565,79.173,179.6445,2.1491,0.0000
C00480=-6.894,54.819,76.901,-170.1659,-10.7275,0.0000
C00481=-3.885,53.739,75.988,-153.1141,-3.8747,0.0000
C00482=-1.568,53.762,75.948,-151.9022,1.0587,0.0000
C00483=0.000,53.776,75.975,-151.8999,-0.0000,0.0000
C00484=0.000,52.771,77.932,-153.7424,-0.0000,0.0000
C00485=1.476,52.759,77.904,-153.7399,-0.9264,0.0000
C00486=3.730,52.747,77.945,-154.9907,3.8073,0.0000
C00487=6.711,53.894,78.888,-171.3661,9.7395,0.0000
C00488=7.974,57.808,81.229,179.6675,-2.0918,0.0000
C00489=8.774,64.206,84.354,179.5984,-2.8375,0.0000
C00490=9.737,72.291,87.405,179.6271,-2.7514,0.0000
C00491=10.790,80.844,89.614,179.6616,-2.5105,0.0000
C00492=11.935,88.455,90.663,179.3521,-2.0976,0.0000
C00493=15.553,93.978,91.206,179.0086,-0.8482,0.0000
C00494=21.285,96.677,91.642,179.4213,-0.0974,0.0000
C00495=27.936,96.017,92.077,179.9656,0.0115,0.0000
C00496=34.820,93.742,92.362,179.9943,0.0000,0.0000
C00497=41.664,90.907,92.362,179.9943,0.0000,0.0000
C00498=48.140,87.648,92.077,179.9656,0.0172,0.0000
C00499=53.310,83.412,91.642,179.6619,0.4813,0.0000
C00500=55.455,77.451,91.206,179.8968,1.3008,0.0000
C00501=54.108,70.986,90.663,-178.9795,1.9429,0.0000
C00502=49.536,64.795,89.614,-178.4633,2.0123,0.0000
C00503=44.233,58.003,87.405,-178.3197,2.2074,0.0000
C00504=39.197,51.604,84.354,-178.2737,2.2936,0.0000
C00505=35.238,46.514,81.229,-178.7503,1.7138,0.0000
C00506=33.363,42.854,78.888,179.2006,-12.8812,0.0000
C00507=34.660,39.935,77.945,-164.2103,-20.6545,0.0000
C00508=36.262,38.350,77.904,-160.1848,-18.6417,0.0000
C00509=37.314,37.314,77.932,-160.7714,-19.2286,0.0000
C00510=38.350,36.262,77.904,-161.3583,-19.8152,0.0000
C00511=39.935,34.660,77.945,-159.3455,-15.7897,0.0000
C00512=42.854,33.363,78.888,-167.1188,0.8053,0.0000
C00513=46.514,35.238,81.229,178.2862,-1.2497,0.0000
C00514=51.604,39.197,84.354,177.7064,-1.7263,0.0000
C00515=58.003,44.233,87.405,177.7926,-1.6803,0.0000
C00516=64.795,49.536,89.614,177.9877,-1.5367,0.0000
C00517=70.986,54.108,90.663,178.0571,-1.0205,0.0000
C00518=77.451,55.455,91.206,178.6992,0.1032,0.0000
C00519=83.412,53.310,91.642,179.5187,0.3381,0.0000
C00520=87.648,48.140,92.077,179.9828,0.0344,0.0000
C00521=90.907,41.664,92.362,180.0000,0.0057,0.0000
C00522=93.742,34.820,92.362,180.0000,0.0057,0.0000
C00523=96.017,27.936,92.077,179.9885,0.0344,0.0000
C00524=96.677,21.285,91.642,-179.9026,0.5787,0.0000
C00525=93.978,15.553,91.206,-179.1518,0.9914,0.0000
C00526=88.455,11.935,90.663,-177.9024,0.6479,0.0000
C00527=80.844,10.790,89.614,-177.4895,0.3384,0.0000
C00528=72.291,9.737,87.405,-177.2486,0.3729,0.0000
C00529=64.206,8.774,84.354,-177.1625,0.4016,0.0000
C00530=57.808,7.974,81.229,-177.9082,0.3325,0.0000
C00531=53.894,6.711,78.888,170.2605,-8.6339,0.0000
C00532=52.747,3.730,77.945,176.1927,-25.0093,0.0000
C00533=52.759,1.476,77.904,-179.0736,-26.2601,0.0000
C00534=52.771,0.000,77.932,-180.0000,-26.2576,0.0000
C00535=52.759,-1.476,77.904,179.0736,-26.2601,0.0000
C00536=52.747,-3.730,77.945,-176.1863,-25.0093,0.0000
C00537=53.894,-6.711,78.888,-170.2605,-8.6339,0.0000
C00538=57.808,-7.974,81.229,177.9082,0.3325,0.0000
C00539=64.206,-8.774,84.354,177.1625,0.4016,0.0000
C00540=72.291,-9.737,87.405,177.2486,0.3729,0.0000
C00541=80.844,-10.790,89.614,177.4895,0.3384,0.0000
C00542=88.455,-11.935,90.663,177.9024,0.6479,0.0000
C00543=93.978,-15.553,91.206,179.1518,0.9914,0.0000
C00544=96.677,-21.285,91.642,179.9026,0.5787,0.0000
C00545=96.017,-27.936,92.077,-179.9885,0.0344,0.0000
C00546=93.742,-34.820,92.362,-180.0000,0.0057,0.0000
C00547=90.907,-41.664,92.362,-180.0000,0.0057,0.0000
C00548=87.648,-48.140,92.077,-179.9828,0.0344,0.0000
C00549=83.412,-53.310,91.642,-179.5187,0.3381,0.0000
C00550=77.451,-55.455,91.206,-178.6992,0.1032,0.0000
C00551=70.986,-54.108,90.663,-178.0571,-1.0205,0.0000
C00552=64.795,-49.536,89.614,-177.9877,-1.5367,0.0000
C00553=58.003,-44.233,87.405,-177.7926,-1.6803,0.0000
C00554=51.604,-39.197,84.354,-177.7064,-1.7263,0.0000
C00555=46.514,-35.238,81.229,-178.2862,-1.2497,0.0000
C00556=42.854,-33.363,78.888,167.1188,0.7994,0.0000
C00557=39.935,-34.660,77.945,159.3455,-15.7897,0.0000
C00558=38.350,-36.262,77.904,161.3583,-19.8152,0.0000
C00559=37.314,-37.314,77.932,160.7714,-19.2286,0.0000
C00560=36.262,-38.350,77.904,160.1848,-18.6417,0.0000
C00561=34.660,-39.935,77.945,164.2103,-20.6545,0.0000
C00562=33.363,-42.854,78.888,-179.1947,-12.8812,0.0000
C00563=35.238,-46.514,81.229,178.7503,1.7138,0.0000
C00564=39.197,-51.604,84.354,178.2737,2.2936,0.0000
C00565=44.233,-58.003,87.405,178.3197,2.2074,0.0000
C00566=49.536,-64.795,89.614,178.4633,2.0123,0.0000
C00567=54.108,-70.986,90.663,178.9795,1.9429,0.0000
C00568=55.455,-77.451,91.206,-179.8968,1.3008,0.0000
C00569=53.310,-83.412,91.642,-179.6619,0.4813,0.0000
C00570=48.140,-87.648,92.077,-179.9656,0.0172,0.0000
C00571=41.664,-90.907,92.362,-179.9943,0.0000,0.0000
C00572=34.820,-93.742,92.362,-179.9943,0.0000,0.0000
C00573=27.936,-96.017,92.077,-179.9656,0.0115,0.0000
C00574=21.285,-96.677,91.642,-179.4213,-0.0974,0.0000
C00575=15.553,-93.978,91.206,-179.0086,-0.8482,0.0000
C00576=11.935,-88.455,90.663,-179.3521,-2.0976,0.0000
C00577=10.790,-80.844,89.614,-179.6616,-2.5105,0.0000
C00578=9.737,-72.291,87.405,-179.6271,-2.7514,0.0000
C00579=8.774,-64.206,84.354,-179.5984,-2.8375,0.0000
C00580=7.974,-57.808,81.229,-179.6675,-2.0918,0.0000
C00581=6.711,-53.894,78.888,171.3661,9.7395,0.0000
C00582=3.730,-52.747,77.945,154.9907,3.8073,0.0000
C00583=1.476,-52.759,77.904,153.7399,-0.9264,0.0000
C00584=0.000,-52.771,77.932,153.7424,-0.0000,0.0000
C00585=0.000,-52.771,77.932,153.7424,-0.0000,0.0000
C00586=-1.476,-52.759,77.904,153.7399,0.9264,0.0000
C00587=-3.730,-52.747,77.945,154.9907,-3.8137,0.0000
C00588=-6.711,-53.894,78.888,171.3661,-9.7395,0.0000
C00589=-7.974,-57.808,81.229,-179.6675,2.0918,0.0000
C00590=-8.774,-64.206,84.354,-179.5984,2.8375,0.0000
C00591=-9.737,-72.291,87.405,-179.6271,2.7514,0.0000
C00592=-10.790,-80.844,89.614,-179.6616,2.5105,0.0000
C00593=-11.935,-88.455,90.663,-179.3521,2.0976,0.0000
C00594=-15.553,-93.978,91.206,-179.0086,0.8482,0.0000
C00595=-21.285,-96.677,91.642,-179.4213,0.0974,0.0000
C00596=-27.936,-96.017,92.077,-179.9656,-0.0115,0.0000
C00597=-34.820,-93.742,92.362,-179.9943,-0.0000,0.0000
C00598=-41.664,-90.907,92.362,-179.9943,-0.0000,0.0000
C00599=-48.140,-87.648,92.077,-179.9656,-0.0172,0.0000
C00600=-53.310,-83.412,91.642,-179.6619,-0.4813,0.0000
C00601=-55.455,-77.451,91.206,-179.8968,-1.3008,0.0000
C00602=-54.108,-70.986,90.663,178.9795,-1.9429,0.0000
C00603=-49.536,-64.795,89.614,178.4633,-2.0123,0.0000
C00604=-44.233,-58.003,87.405,178.3197,-2.2074,0.0000
C00605=-39.197,-51.604,84.354,178.2737,-2.2936,0.0000
C00606=-35.238,-46.514,81.229,178.7503,-1.7138,0.0000
C00607=-33.363,-42.854,78.888,-179.2006,12.8812,0.0000
C00608=-34.660,-39.935,77.945,164.2103,20.6545,0.0000
C00609=-36.262,-38.350,77.904,160.1848,18.6417,0.0000
C00610=-37.314,-37.314,77.932,160.7714,19.2286,0.0000
C00611=-38.350,-36.262,77.904,161.3583,19.8152,0.0000
C00612=-39.935,-34.660,77.945,159.3455,15.7897,0.0000
C00613=-42.854,-33.363,78.888,167.1188,-0.8053,0.0000
C00614=-46.514,-35.238,81.229,-178.2862,1.2497,0.0000
C00615=-51.604,-39.197,84.354,-177.7064,1.7263,0.0000
C00616=-58.003,-44.233,87.405,-177.7926,1.6803,0.0000
C00617=-64.795,-49.536,89.614,-177.9877,1.5367,0.0000
C00618=-70.986,-54.108,90.663,-178.0571,1.0205,0.0000
C00619=-77.451,-55.455,91.206,-178.6992,-0.1032,0.0000
C00620=-83.412,-53.310,91.642,-179.5187,-0.3381,0.0000
C00621=-87.648,-48.140,92.077,-179.9828,-0.0344,0.0000
C00622=-90.907,-41.664,92.362,-180.0000,-0.0057,0.0000
C00623=-93.742,-34.820,92.362,-180.0000,-0.0057,0.0000
C00624=-96.017,-27.936,92.077,-179.9885,-0.0344,0.0000
C00625=-96.677,-21.285,91.642,179.9026,-0.5787,0.0000
C00626=-93.978,-15.553,91.206,179.1518,-0.9914,0.0000
C00627=-88.455,-11.935,90.663,177.9024,-0.6479,0.0000
C00628=-80.844,-10.790,89.614,177.4895,-0.3384,0.0000
C00629=-72.291,-9.737,87.405,177.2486,-0.3729,0.0000
C00630=-64.206,-8.774,84.354,177.1625,-0.4016,0.0000
C00631=-57.808,-7.974,81.229,177.9082,-0.3325,0.0000
C00632=-53.894,-6.711,78.888,-170.2605,8.6339,0.0000
C00633=-52.747,-3.730,77.945,-176.1927,25.0093,0.0000
C00634=-52.759,-1.476,77.904,179.0736,26.2601,0.0000
C00635=-52.771,0.000,77.932,180.0000,26.2576,0.0000
C00636=-52.759,1.476,77.904,-179.0736,26.2601,0.0000
C00637=-52.747,3.730,77.945,176.1863,25.0093,0.0000
C00638=-53.894,6.711,78.888,170.2605,8.6339,0.0000
C00639=-57.808,7.974,81.229,-177.9082,-0.3325,0.0000
C00640=-64.206,8.774,84.354,-177.1625,-0.4016,0.0000
C00641=-72.291,9.737,87.405,-177.2486,-0.3729,0.0000
C00642=-80.844,10.790,89.614,-177.4895,-0.3384,0.0000
C00643=-88.455,11.935,90.663,-177.9024,-0.6479,0.0000
C00644=-93.978,15.553,91.206,-179.1518,-0.9914,0.0000
C00645=-96.677,21.285,91.642,-179.9026,-0.5787,0.0000
C00646=-96.017,27.936,92.077,179.9885,-0.0344,0.0000
C00647=-93.742,34.820,92.362,180.0000,-0.0057,0.0000
C00648=-90.907,41.664,92.362,180.0000,-0.0057,0.0000
C00649=-87.648,48.140,92.077,179.9828,-0.0344,0.0000
C00650=-83.412,53.310,91.642,179.5187,-0.3381,0.0000
C00651=-77.451,55.455,91.206,178.6992,-0.1032,0.0000
C00652=-70.986,54.108,90.663,178.0571,1.0205,0.0000
C00653=-64.795,49.536,89.614,177.9877,1.5367,0.0000
C00654=-58.003,44.233,87.405,177.7926,1.6803,0.0000
C00655=-51.604,39.197,84.354,177.7064,1.7263,0.0000
C00656=-46.514,35.238,81.229,178.2862,1.2497,0.0000
C00657=-42.854,33.363,78.888,-167.1188,-0.7994,0.0000
C00658=-39.935,34.660,77.945,-159.3455,15.7897,0.0000
C00659=-38.350,36.262,77.904,-161.3583,19.8152,0.0000
C00660=-37.314,37.314,77.932,-160.7714,19.2286,0.0000
C00661=-36.262,38.350,77.904,-160.1848,18.6417,0.0000
C00662=-34.660,39.935,77.945,-164.2103,20.6545,0.0000
C00663=-33.363,42.854,78.888,179.1947,12.8812,0.0000
C00664=-35.238,46.514,81.229,-178.7503,-1.7138,0.0000
C00665=-39.197,51.604,84.354,-178.2737,-2.2936,0.0000
C00666=-44.233,58.003,87.405,-178.3197,-2.2074,0.0000
C00667=-49.536,64.795,89.614,-178.4633,-2.0123,0.0000
C00668=-54.108,70.986,90.663,-178.9795,-1.9429,0.0000
C00669=-55.455,77.451,91.206,179.8968,-1.3008,0.0000
C00670=-53.310,83.412,91.642,179.6619,-0.4813,0.0000
C00671=-48.140,87.648,92.077,179.9656,-0.0172,0.0000
C00672=-41.664,90.907,92.362,179.9943,-0.0000,0.0000
C00673=-34.820,93.742,92.362,179.9943,-0.0000,0.0000
C00674=-27.936,96.017,92.077,179.9656,-0.0115,0.0000
C00675=-21.285,96.677,91.642,179.4213,0.0974,0.0000
C00676=-15.553,93.978,91.206,179.0086,0.8482,0.0000
C00677=-11.935,88.455,90.663,179.3521,2.0976,0.0000
C00678=-10.790,80.844,89.614,179.6616,2.5105,0.0000
C00679=-9.737,72.291,87.405,179.6271,2.7514,0.0000
C00680=-8.774,64.206,84.354,179.5984,2.8375,0.0000
C00681=-7.974,57.808,81.229,179.6675,2.0918,0.0000
C00682=-6.711,53.894,78.888,-171.3661,-9.7395,0.0000
C00683=-3.730,52.747,77.945,-154.9907,-3.8137,0.0000
C00684=-1.476,52.759,77.904,-153.7399,0.9264,0.0000
C00685=0.000,52.771,77.932,-153.7424,-0.0000,0.0000
C00686=0.000,51.832,79.921,-155.8007,-0.0000,0.0000
C00687=1.391,51.822,79.893,-155.7984,-0.7978,0.0000
C00688=3.586,51.820,79.935,-157.0592,3.6722,0.0000
C00689=6.543,53.038,80.908,-172.5264,8.6939,0.0000
C00690=7.793,57.125,83.313,179.7019,-1.9657,0.0000
C00691=8.610,63.749,86.500,179.6674,-2.4072,0.0000
C00692=9.608,72.041,89.587,179.7191,-2.1147,0.0000
C00693=10.692,80.728,91.809,179.7765,-1.6904,0.0000
C00694=11.850,88.408,92.861,179.6103,-1.2664,0.0000
C00695=15.484,93.970,93.405,179.4499,-0.4699,0.0000
C00696=21.237,96.685,93.841,179.7078,-0.0516,0.0000
C00697=27.910,96.026,94.277,179.9828,0.0057,0.0000
C00698=34.811,93.745,94.562,180.0000,0.0000,0.0000
C00699=41.672,90.903,94.562,180.0000,0.0000,0.0000
C00700=48.166,87.636,94.277,179.9885,0.0057,0.0000
C00701=53.350,83.383,93.841,179.8281,0.2464,0.0000
C00702=55.498,77.395,93.405,179.9427,0.7220,0.0000
C00703=54.135,70.893,92.861,-179.3810,1.1690,0.0000
C00704=49.523,64.644,91.809,-178.9626,1.3525,0.0000
C00705=44.146,57.735,89.587,-178.7044,1.6966,0.0000
C00706=38.990,51.166,86.500,-178.5322,1.9376,0.0000
C00707=34.883,45.903,83.313,-178.8192,1.5991,0.0000
C00708=32.877,42.130,80.908,179.1175,-11.3627,0.0000
C00709=34.107,39.178,79.935,-165.7484,-19.0145,0.0000
C00710=35.661,37.627,79.893,-161.8596,-17.1191,0.0000
C00711=36.651,36.651,79.921,-162.3735,-17.6265,0.0000
C00712=37.627,35.661,79.893,-162.8809,-18.1461,0.0000
C00713=39.178,34.107,79.935,-160.9800,-14.2458,0.0000
C00714=42.130,32.877,80.908,-168.6373,0.8825,0.0000
C00715=45.903,34.883,83.313,178.4009,-1.1808,0.0000
C00716=51.166,38.990,86.500,178.0624,-1.4678,0.0000
C00717=57.735,44.146,89.587,178.3034,-1.2956,0.0000
C00718=64.644,49.523,91.809,178.6475,-1.0374,0.0000
C00719=70.893,54.135,92.861,178.8310,-0.6190,0.0000
C00720=77.395,55.498,93.405,179.2780,0.0573,0.0000
C00721=83.383,53.350,93.841,179.7536,0.1719,0.0000
C00722=87.636,48.166,94.277,179.9943,0.0115,0.0000
C00723=90.903,41.672,94.562,180.0000,0.0000,0.0000
C00724=93.745,34.811,94.562,180.0000,0.0000,0.0000
C00725=96.026,27.910,94.277,179.9943,0.0172,0.0000
C00726=96.685,21.237,93.841,-179.9484,0.2922,0.0000
C00727=93.970,15.484,93.405,-179.5301,0.5501,0.0000
C00728=88.408,11.850,92.861,-178.7336,0.3897,0.0000
C00729=80.728,10.692,91.809,-178.3096,0.2235,0.0000
C00730=72.041,9.608,89.587,-177.8853,0.2809,0.0000
C00731=63.749,8.610,86.500,-177.5928,0.3326,0.0000
C00732=57.125,7.793,83.313,-178.0343,0.2981,0.0000
C00733=53.038,6.543,80.908,171.3061,-7.4736,0.0000
C00734=51.820,3.586,79.935,176.3278,-22.9408,0.0000
C00735=51.822,1.391,79.893,-179.2022,-24.2016,0.0000
C00736=51.832,0.000,79.921,-180.0000,-24.1993,0.0000
C00737=51.822,-1.390,79.893,179.2022,-24.2016,0.0000
C00738=51.820,-3.586,79.935,-176.3278,-22.9408,0.0000
C00739=53.038,-6.543,80.908,-171.3061,-7.4736,0.0000
C00740=57.125,-7.793,83.313,178.0343,0.2981,0.0000
C00741=63.749,-8.610,86.500,177.5928,0.3326,0.0000
C00742=72.041,-9.608,89.587,177.8853,0.2809,0.0000
C00743=80.728,-10.692,91.809,178.3096,0.2235,0.0000
C00744=88.408,-11.850,92.861,178.7336,0.3897,0.0000
C00745=93.970,-15.484,93.405,179.5301,0.5501,0.0000
C00746=96.685,-21.237,93.841,179.9484,0.2922,0.0000
C00747=96.026,-27.910,94.277,-179.9943,0.0172,0.0000
C00748=93.745,-34.811,94.562,-180.0000,0.0000,0.0000
C00749=90.903,-41.672,94.562,-180.0000,0.0000,0.0000
C00750=87.636,-48.166,94.277,-179.9943,0.0115,0.0000
C00751=83.383,-53.350,93.841,-179.7536,0.1719,0.0000
C00752=77.395,-55.498,93.405,-179.2780,0.0573,0.0000
C00753=70.893,-54.135,92.861,-178.8310,-0.6190,0.0000
C00754=64.644,-49.523,91.809,-178.6475,-1.0374,0.0000
C00755=57.735,-44.146,89.587,-178.3034,-1.2956,0.0000
C00756=51.166,-38.990,86.500,-178.0624,-1.4678,0.0000
C00757=45.903,-34.883,83.313,-178.4009,-1.1808,0.0000
C00758=42.130,-32.877,80.908,168.6373,0.8825,0.0000
C00759=39.178,-34.107,79.935,160.9855,-14.2516,0.0000
C00760=37.627,-35.661,79.893,162.8809,-18.1404,0.0000
C00761=36.651,-36.651,79.921,162.3735,-17.6265,0.0000
C00762=35.661,-37.627,79.893,161.8539,-17.1191,0.0000
C00763=34.107,-39.178,79.935,165.7542,-19.0200,0.0000
C00764=32.877,-42.130,80.908,-179.1175,-11.3627,0.0000
C00765=34.883,-45.903,83.313,178.8192,1.5991,0.0000
C00766=38.990,-51.166,86.500,178.5322,1.9376,0.0000
C00767=44.146,-57.735,89.587,178.7044,1.6966,0.0000
C00768=49.523,-64.644,91.809,178.9626,1.3525,0.0000
C00769=54.135,-70.893,92.861,179.3810,1.1690,0.0000
C00770=55.498,-77.395,93.405,-179.9427,0.7220,0.0000
C00771=53.350,-83.383,93.841,-179.8281,0.2464,0.0000
C00772=48.166,-87.636,94.277,-179.9885,0.0057,0.0000
C00773=41.672,-90.903,94.562,-180.0000,0.0000,0.0000
C00774=34.811,-93.745,94.562,-180.0000,0.0000,0.0000
C00775=27.910,-96.026,94.277,-179.9828,0.0057,0.0000
C00776=21.237,-96.685,93.841,-179.7078,-0.0516,0.0000
C00777=15.484,-93.970,93.405,-179.4499,-0.4699,0.0000
C00778=11.850,-88.408,92.861,-179.6103,-1.2664,0.0000
C00779=10.692,-80.728,91.809,-179.7765,-1.6904,0.0000
C00780=9.608,-72.041,89.587,-179.7191,-2.1147,0.0000
C00781=8.610,-63.749,86.500,-179.6674,-2.4072,0.0000
C00782=7.793,-57.125,83.313,-179.7019,-1.9657,0.0000
C00783=6.543,-53.038,80.908,172.5264,8.6939,0.0000
C00784=3.586,-51.820,79.935,157.0592,3.6722,0.0000
C00785=1.391,-51.822,79.893,155.7984,-0.7978,0.0000
C00786=0.000,-51.832,79.921,155.8007,-0.0000,0.0000
C00787=0.000,-51.832,79.921,155.8007,-0.0000,0.0000
C00788=-1.390,-51.822,79.893,155.7984,0.7978,0.0000
C00789=-3.586,-51.820,79.935,157.0592,-3.6722,0.0000
C00790=-6.543,-53.038,80.908,172.5264,-8.6939,0.0000
C00791=-7.793,-57.125,83.313,-179.7019,1.9657,0.0000
C00792=-8.610,-63.749,86.500,-179.6674,2.4072,0.0000
C00793=-9.608,-72.041,89.587,-179.7191,2.1147,0.0000
C00794=-10.692,-80.728,91.809,-179.7765,1.6904,0.0000
C00795=-11.850,-88.408,92.861,-179.6103,1.2664,0.0000
C00796=-15.484,-93.970,93.405,-179.4499,0.4699,0.0000
C00797=-21.237,-96.685,93.841,-179.7078,0.0516,0.0000
C00798=-27.910,-96.026,94.277,-179.9828,-0.0057,0.0000
C00799=-34.811,-93.745,94.562,-180.0000,-0.0000,0.0000
C00800=-41.672,-90.903,94.562,-180.0000,-0.0000,0.0000
C00801=-48.166,-87.636,94.277,-179.9885,-0.0057,0.0000
C00802=-53.350,-83.383,93.841,-179.8281,-0.2464,0.0000
C00803=-55.498,-77.395,93.405,-179.9427,-0.7220,0.0000
C00804=-54.135,-70.893,92.861,179.3810,-1.1690,0.0000
C00805=-49.523,-64.644,91.809,178.9626,-1.3525,0.0000
C00806=-44.146,-57.735,89.587,178.7044,-1.6966,0.0000
C00807=-38.990,-51.166,86.500,178.5322,-1.9376,0.0000
C00808=-34.883,-45.903,83.313,178.8192,-1.5991,0.0000
C00809=-32.877,-42.130,80.908,-179.1175,11.3627,0.0000
C00810=-34.107,-39.178,79.935,165.7484,19.0145,0.0000
C00811=-35.661,-37.627,79.893,161.8596,17.1191,0.0000
C00812=-36.651,-36.651,79.921,162.3735,17.6265,0.0000
C00813=-37.627,-35.661,79.893,162.8809,18.1461,0.0000
C00814=-39.178,-34.107,79.935,160.9800,14.2458,0.0000
C00815=-42.130,-32.877,80.908,168.6373,-0.8825,0.0000
C00816=-45.903,-34.883,83.313,-178.4009,1.1808,0.0000
C00817=-51.166,-38.990,86.500,-178.0624,1.4678,0.0000
C00818=-57.735,-44.146,89.587,-178.3034,1.2956,0.0000
C00819=-64.644,-49.523,91.809,-178.6475,1.0374,0.0000
C00820=-70.893,-54.135,92.861,-178.8310,0.6190,0.0000
C00821=-77.395,-55.498,93.405,-179.2780,-0.0573,0.0000
C00822=-83.383,-53.350,93.841,-179.7536,-0.1719,0.0000
C00823=-87.636,-48.166,94.277,-179.9943,-0.0115,0.0000
C00824=-90.903,-41.672,94.562,-180.0000,-0.0000,0.0000
C00825=-93.745,-34.811,94.562,-180.0000,-0.0000,0.0000
C00826=-96.026,-27.910,94.277,-179.9943,-0.0172,0.0000
C00827=-96.685,-21.237,93.841,179.9484,-0.2922,0.0000
C00828=-93.970,-15.484,93.405,179.5301,-0.5501,0.0000
C00829=-88.408,-11.850,92.861,178.7336,-0.3897,0.0000
C00830=-80.728,-10.692,91.809,178.3096,-0.2235,0.0000
C00831=-72.041,-9.608,89.587,177.8853,-0.2809,0.0000
C00832=-63.749,-8.610,86.500,177.5928,-0.3326,0.0000
C00833=-57.125,-7.793,83.313,178.0343,-0.2981,0.0000
C00834=-53.038,-6.543,80.908,-171.3061,7.4736,0.0000
C00835=-51.820,-3.586,79.935,-176.3278,22.9408,0.0000
C00836=-51.822,-1.391,79.893,179.2022,24.2016,0.0000
C00837=-51.832,0.000,79.921,180.0000,24.1993,0.0000
C00838=-51.822,1.390,79.893,-179.2022,24.2016,0.0000
C00839=-51.820,3.586,79.935,176.3278,22.9408,0.0000
C00840=-53.038,6.543,80.908,171.3061,7.4736,0.0000
C00841=-57.125,7.793,83.313,-178.0343,-0.2981,0.0000
C00842=-63.749,8.610,86.500,-177.5928,-0.3326,0.0000
C00843=-72.041,9.608,89.587,-177.8853,-0.2809,0.0000
C00844=-80.728,10.692,91.809,-178.3096,-0.2235,0.0000
C00845=-88.408,11.850,92.861,-178.7336,-0.3897,0.0000
C00846=-93.970,15.484,93.405,-179.5301,-0.5501,0.0000
C00847=-96.685,21.237,93.841,-179.9484,-0.2922,0.0000
C00848=-96.026,27.910,94.277,179.9943,-0.0172,0.0000
C00849=-93.745,34.811,94.562,180.0000,-0.0000,0.0000
C00850=-90.903,41.672,94.562,180.0000,-0.0000,0.0000
C00851=-87.636,48.166,94.277,179.9943,-0.0115,0.0000
C00852=-83.383,53.350,93.841,179.7536,-0.1719,0.0000
C00853=-77.395,55.498,93.405,179.2780,-0.0573,0.0000
C00854=-70.893,54.135,92.861,178.8310,0.6190,0.0000
C00855=-64.644,49.523,91.809,178.6475,1.0374,0.0000
C00856=-57.735,44.146,89.587,178.3034,1.2956,0.0000
C00857=-51.166,38.990,86.500,178.0624,1.4678,0.0000
C00858=-45.903,34.883,83.313,178.4009,1.1808,0.0000
C00859=-42.130,32.877,80.908,-168.6373,-0.8825,0.0000
C00860=-39.178,34.107,79.935,-160.9855,14.2516,0.0000
C00861=-37.627,35.661,79.893,-162.8809,18.1404,0.0000
C00862=-36.651,36.651,79.921,-162.3735,17.6265,0.0000
C00863=-35.661,37.627,79.893,-161.8539,17.1191,0.0000
C00864=-34.107,39.178,79.935,-165.7542,19.0200,0.0000
C00865=-32.877,42.130,80.908,179.1175,11.3627,0.0000
C00866=-34.883,45.903,83.313,-178.8192,-1.5991,0.0000
C00867=-38.990,51.166,86.500,-178.5322,-1.9376,0.0000
C00868=-44.146,57.735,89.587,-178.7044,-1.6966,0.0000
C00869=-49.523,64.644,91.809,-178.9626,-1.3525,0.0000
C00870=-54.135,70.893,92.861,-179.3810,-1.1690,0.0000
C00871=-55.498,77.395,93.405,179.9427,-0.7220,0.0000
C00872=-53.350,83.383,93.841,179.8281,-0.2464,0.0000
C00873=-48.166,87.636,94.277,179.9885,-0.0057,0.0000
C00874=-41.672,90.903,94.562,180.0000,-0.0000,0.0000
C00875=-34.811,93.745,94.562,180.0000,-0.0000,0.0000
C00876=-27.910,96.026,94.277,179.9828,-0.0057,0.0000
C00877=-21.237,96.685,93.841,179.7078,0.0516,0.0000
C00878=-15.484,93.970,93.405,179.4499,0.4699,0.0000
C00879=-11.850,88.408,92.861,179.6103,1.2664,0.0000
C00880=-10.692,80.728,91.809,179.7765,1.6904,0.0000
C00881=-9.608,72.041,89.587,179.7191,2.1147,0.0000
C00882=-8.610,63.749,86.500,179.6674,2.4072,0.0000
C00883=-7.793,57.125,83.313,179.7019,1.9657,0.0000
C00884=-6.543,53.038,80.908,-172.5264,-8.6939,0.0000
C00885=-3.586,51.820,79.935,-157.0592,-3.6722,0.0000
C00886=-1.390,51.822,79.893,-155.7984,0.7978,0.0000
C00887=0.000,51.832,79.921,-155.8007,-0.0000,0.0000
C00888=0.000,50.970,81.946,-158.1007,-0.0000,0.0000
C00889=1.312,50.962,81.916,-158.0911,-0.6670,0.0000
C00890=3.453,50.970,81.960,-159.3378,3.4488,0.0000
C00891=6.389,52.261,82.960,-173.6407,7.6026,0.0000
C00892=7.633,56.525,85.423,179.7420,-1.7650,0.0000
C00893=8.475,63.374,88.663,179.7363,-1.9256,0.0000
C00894=9.515,71.858,91.777,179.8109,-1.4325,0.0000
C00895=10.634,80.658,94.007,179.8911,-0.8251,0.0000
C00896=11.808,88.386,95.061,179.8797,-0.3896,0.0000
C00897=15.455,93.966,95.604,179.9141,-0.0745,0.0000
C00898=55.516,77.372,95.604,179.9943,0.1146,0.0000
C00899=54.149,70.847,95.061,-179.8109,0.3610,0.0000
C00900=49.515,64.553,94.007,-179.4958,0.6589,0.0000
C00901=44.083,57.539,91.777,-179.1232,1.1461,0.0000
C00902=38.820,50.805,88.663,-178.8192,1.5475,0.0000
C00903=34.571,45.367,85.423,-178.9339,1.4271,0.0000
C00904=32.436,41.472,82.960,179.1045,-9.8297,0.0000
C00905=33.599,38.483,81.960,-167.3719,-17.1841,0.0000
C00906=35.108,36.963,81.916,-163.6874,-15.4384,0.0000
C00907=36.041,36.041,81.946,-164.1354,-15.8646,0.0000
C00908=36.963,35.108,81.916,-164.5616,-16.3126,0.0000
C00909=38.483,33.599,81.960,-162.8159,-12.6281,0.0000
C00910=41.472,32.436,82.960,-170.1759,0.8955,0.0000
C00911=45.367,34.571,85.423,178.5729,-1.0661,0.0000
C00912=50.805,38.820,88.663,178.4525,-1.1808,0.0000
C00913=57.539,44.083,91.777,178.8539,-0.8768,0.0000
C00914=64.553,49.515,94.007,179.3411,-0.5042,0.0000
C00915=70.847,54.149,95.061,179.6390,-0.1891,0.0000
C00916=77.372,55.516,95.604,179.8854,0.0057,0.0000
C00917=93.966,15.455,95.604,-179.9255,0.0859,0.0000
C00918=88.386,11.808,95.061,-179.6104,0.1203,0.0000
C00919=80.658,10.634,94.007,-179.1749,0.1089,0.0000
C00920=71.858,9.515,91.777,-178.5675,0.1891,0.0000
C00921=63.374,8.475,88.663,-178.0744,0.2637,0.0000
C00922=56.525,7.633,85.423,-178.2350,0.2580,0.0000
C00923=52.261,6.389,82.960,172.3974,-6.3593,0.0000
C00924=50.970,3.453,81.960,176.5512,-20.6622,0.0000
C00925=50.962,1.312,81.916,-179.3330,-21.9089,0.0000
C00926=50.970,0.000,81.946,-180.0000,-21.8993,0.0000
C00927=50.962,-1.311,81.916,179.3330,-21.9089,0.0000
C00928=50.970,-3.454,81.960,-176.5512,-20.6622,0.0000
C00929=52.261,-6.389,82.960,-172.3974,-6.3593,0.0000
C00930=56.525,-7.633,85.423,178.2350,0.2580,0.0000
C00931=63.374,-8.475,88.663,178.0744,0.2637,0.0000
C00932=71.858,-9.515,91.777,178.5675,0.1891,0.0000
C00933=80.658,-10.634,94.007,179.1749,0.1089,0.0000
C00934=88.386,-11.808,95.061,179.6104,0.1203,0.0000
C00935=93.966,-15.455,95.604,179.9255,0.0859,0.0000
C00936=77.372,-55.516,95.604,-179.8854,0.0057,0.0000
C00937=70.847,-54.149,95.061,-179.6390,-0.1891,0.0000
C00938=64.553,-49.515,94.007,-179.3411,-0.5042,0.0000
C00939=57.539,-44.083,91.777,-178.8539,-0.8768,0.0000
C00940=50.805,-38.820,88.663,-178.4525,-1.1808,0.0000
C00941=45.367,-34.571,85.423,-178.5729,-1.0661,0.0000
C00942=41.472,-32.436,82.960,170.1703,0.8955,0.0000
C00943=38.483,-33.599,81.960,162.8159,-12.6281,0.0000
C00944=36.963,-35.108,81.916,164.5616,-16.3126,0.0000
C00945=36.041,-36.041,81.946,164.1354,-15.8646,0.0000
C00946=35.108,-36.963,81.916,163.6874,-15.4384,0.0000
C00947=33.599,-38.483,81.960,167.3719,-17.1841,0.0000
C00948=32.436,-41.472,82.960,-179.1045,-9.8241,0.0000
C00949=34.571,-45.367,85.423,178.9339,1.4271,0.0000
C00950=38.820,-50.805,88.663,178.8192,1.5475,0.0000
C00951=44.083,-57.539,91.777,179.1232,1.1461,0.0000
C00952=49.515,-64.553,94.007,179.4958,0.6589,0.0000
C00953=54.149,-70.847,95.061,179.8109,0.3610,0.0000
C00954=55.516,-77.372,95.604,-179.9943,0.1146,0.0000
C00955=15.455,-93.966,95.604,-179.9141,-0.0745,0.0000
C00956=11.808,-88.386,95.061,-179.8797,-0.3896,0.0000
C00957=10.634,-80.658,94.007,-179.8911,-0.8251,0.0000
C00958=9.515,-71.858,91.777,-179.8109,-1.4325,0.0000
C00959=8.475,-63.374,88.663,-179.7363,-1.9256,0.0000
C00960=7.633,-56.525,85.423,-179.7420,-1.7650,0.0000
C00961=6.389,-52.261,82.960,173.6407,7.6026,0.0000
C00962=3.453,-50.970,81.960,159.3378,3.4488,0.0000
C00963=1.312,-50.962,81.916,158.0911,-0.6670,0.0000
C00964=0.000,-50.970,81.946,158.1007,-0.0000,0.0000
C00965=0.000,-50.970,81.946,158.1007,-0.0000,0.0000
C00966=-1.311,-50.962,81.916,158.0911,0.6670,0.0000
C00967=-3.454,-50.970,81.960,159.3378,-3.4488,0.0000
C00968=-6.389,-52.261,82.960,173.6407,-7.6026,0.0000
C00969=-7.633,-56.525,85.423,-179.7420,1.7650,0.0000
C00970=-8.475,-63.374,88.663,-179.7363,1.9256,0.0000
C00971=-9.515,-71.858,91.777,-179.8109,1.4325,0.0000
C00972=-10.634,-80.658,94.007,-179.8911,0.8251,0.0000
C00973=-11.808,-88.386,95.061,-179.8797,0.3896,0.0000
C00974=-15.455,-93.966,95.604,-179.9141,0.0745,0.0000
C00975=-55.516,-77.372,95.604,-179.9943,-0.1146,0.0000
C00976=-54.149,-70.847,95.061,179.8109,-0.3610,0.0000
C00977=-49.515,-64.553,94.007,179.4958,-0.6589,0.0000
C00978=-44.083,-57.539,91.777,179.1232,-1.1461,0.0000
C00979=-38.820,-50.805,88.663,178.8192,-1.5475,0.0000
C00980=-34.571,-45.367,85.423,178.9339,-1.4271,0.0000
C00981=-32.436,-41.472,82.960,-179.1045,9.8297,0.0000
C00982=-33.599,-38.483,81.960,167.3719,17.1841,0.0000
C00983=-35.108,-36.963,81.916,163.6874,15.4384,0.0000
C00984=-36.041,-36.041,81.946,164.1354,15.8646,0.0000
C00985=-36.963,-35.108,81.916,164.5616,16.3126,0.0000
C00986=-38.483,-33.599,81.960,162.8159,12.6281,0.0000
C00987=-41.472,-32.436,82.960,170.1759,-0.8955,0.0000
C00988=-45.367,-34.571,85.423,-178.5729,1.0661,0.0000
C00989=-50.805,-38.820,88.663,-178.4525,1.1808,0.0000
C00990=-57.539,-44.083,91.777,-178.8539,0.8768,0.0000
C00991=-64.553,-49.515,94.007,-179.3411,0.5042,0.0000
C00992=-70.847,-54.149,95.061,-179.6390,0.1891,0.0000
C00993=-77.372,-55.516,95.604,-179.8854,-0.0057,0.0000
C00994=-93.966,-15.455,95.604,179.9255,-0.0859,0.0000
C00995=-88.386,-11.808,95.061,179.6104,-0.1203,0.0000
C00996=-80.658,-10.634,94.007,179.1749,-0.1089,0.0000
C00997=-71.858,-9.515,91.777,178.5675,-0.1891,0.0000
C00998=-63.374,-8.475,88.663,178.0744,-0.2637,0.0000
C00999=-56.525,-7.633,85.423,178.2350,-0.2580,0.0000
C01000=-52.261,-6.389,82.960,-172.3974,6.3593,0.0000
C01001=-50.970,-3.453,81.960,-176.5512,20.6622,0.0000
C01002=-50.962,-1.312,81.916,179.3330,21.9089,0.0000
C01003=-50.970,0.000,81.946,180.0000,21.8993,0.0000
C01004=-50.962,1.311,81.916,-179.3330,21.9089,0.0000
C01005=-50.970,3.454,81.960,176.5512,20.6622,0.0000
C01006=-52.261,6.389,82.960,172.3974,6.3593,0.0000
C01007=-56.525,7.633,85.423,-178.2350,-0.2580,0.0000
C01008=-63.374,8.475,88.663,-178.0744,-0.2637,0.0000
C01009=-71.858,9.515,91.777,-178.5675,-0.1891,0.0000
C01010=-80.658,10.634,94.007,-179.1749,-0.1089,0.0000
C01011=-88.386,11.808,95.061,-179.6104,-0.1203,0.0000
C01012=-93.966,15.455,95.604,-179.9255,-0.0859,0.0000
C01013=-77.372,55.516,95.604,179.8854,-0.0057,0.0000
C01014=-70.847,54.149,95.061,179.6390,0.1891,0.0000
C01015=-64.553,49.515,94.007,179.3411,0.5042,0.0000
C01016=-57.539,44.083,91.777,178.8539,0.8768,0.0000
C01017=-50.805,38.820,88.663,178.4525,1.1808,0.0000
C01018=-45.367,34.571,85.423,178.5729,1.0661,0.0000
C01019=-41.472,32.436,82.960,-170.1703,-0.8955,0.0000
C01020=-38.483,33.599,81.960,-162.8159,12.6281,0.0000
C01021=-36.963,35.108,81.916,-164.5616,16.3126,0.0000
C01022=-36.041,36.041,81.946,-164.1354,15.8646,0.0000
C01023=-35.108,36.963,81.916,-163.6874,15.4384,0.0000
C01024=-33.599,38.483,81.960,-167.3719,17.1841,0.0000
C01025=-32.436,41.472,82.960,179.1045,9.8241,0.0000
C01026=-34.571,45.367,85.423,-178.9339,-1.4271,0.0000
C01027=-38.820,50.805,88.663,-178.8192,-1.5475,0.0000
C01028=-44.083,57.539,91.777,-179.1232,-1.1461,0.0000
C01029=-49.515,64.553,94.007,-179.4958,-0.6589,0.0000
C01030=-54.149,70.847,95.061,-179.8109,-0.3610,0.0000
C01031=-55.516,77.372,95.604,179.9943,-0.1146,0.0000
C01032=-15.455,93.966,95.604,179.9141,0.0745,0.0000
C01033=-11.808,88.386,95.061,179.8797,0.3896,0.0000
C01034=-10.634,80.658,94.007,179.8911,0.8251,0.0000
C01035=-9.515,71.858,91.777,179.8109,1.4325,0.0000
C01036=-8.475,63.374,88.663,179.7363,1.9256,0.0000
C01037=-7.633,56.525,85.423,179.7420,1.7650,0.0000
C01038=-6.389,52.261,82.960,-173.6407,-7.6026,0.0000
C01039=-3.454,50.970,81.960,-159.3378,-3.4488,0.0000
C01040=-1.311,50.962,81.916,-158.0911,0.6670,0.0000
C01041=0.000,50.970,81.946,-158.1007,-0.0000,0.0000
C01042=0.000,50.195,84.004,-160.6645,-0.0000,0.0000
C01043=1.241,50.188,83.974,-160.6464,-0.5465,0.0000
C01044=3.334,50.204,84.019,-161.8426,3.1427,0.0000
C01045=6.253,51.571,85.045,-174.7226,6.4692,0.0000
C01046=7.499,56.017,87.559,179.7879,-1.5013,0.0000
C01047=8.371,63.087,90.842,179.8109,-1.3982,0.0000
C01048=9.459,71.748,93.974,179.9083,-0.7048,0.0000
C01049=44.045,57.421,93.974,-179.5702,0.5615,0.0000
C01050=38.690,50.529,90.842,-179.1404,1.1232,0.0000
C01051=34.307,44.912,87.559,-179.0888,1.2091,0.0000
C01052=32.045,40.888,85.045,179.1489,-8.2800,0.0000
C01053=33.142,37.857,84.019,-169.0726,-15.1488,0.0000
C01054=34.611,36.365,83.974,-165.6883,-13.5853,0.0000
C01055=35.493,35.493,84.004,-166.0610,-13.9333,0.0000
C01056=36.365,34.611,83.974,-166.4147,-14.3117,0.0000
C01057=37.858,33.142,84.019,-164.8512,-10.9274,0.0000
C01058=40.888,32.045,85.045,-171.7200,0.8511,0.0000
C01059=44.912,34.307,87.559,178.7909,-0.9112,0.0000
C01060=50.529,38.690,90.842,178.8768,-0.8596,0.0000
C01061=57.421,44.045,93.974,179.4385,-0.4298,0.0000
C01062=71.748,9.459,93.974,-179.2952,0.0917,0.0000
C01063=63.087,8.371,90.842,-178.6018,0.1891,0.0000
C01064=56.017,7.499,87.559,-178.4987,0.2121,0.0000
C01065=51.571,6.253,85.045,173.5308,-5.2774,0.0000
C01066=50.204,3.334,84.019,176.8573,-18.1574,0.0000
C01067=50.188,1.241,83.974,-179.4535,-19.3536,0.0000
C01068=50.195,0.000,84.004,-180.0000,-19.3355,0.0000
C01069=50.188,-1.240,83.974,179.4535,-19.3536,0.0000
C01070=50.204,-3.335,84.019,-176.8573,-18.1574,0.0000
C01071=51.571,-6.253,85.045,-173.5308,-5.2774,0.0000
C01072=56.017,-7.499,87.559,178.4987,0.2121,0.0000
C01073=63.087,-8.371,90.842,178.6018,0.1891,0.0000
C01074=71.748,-9.459,93.974,179.2952,0.0917,0.0000
C01075=57.421,-44.045,93.974,-179.4385,-0.4298,0.0000
C01076=50.529,-38.690,90.842,-178.8768,-0.8596,0.0000
C01077=44.912,-34.307,87.559,-178.7909,-0.9112,0.0000
C01078=40.888,-32.045,85.045,171.7200,0.8511,0.0000
C01079=37.857,-33.142,84.019,164.8512,-10.9274,0.0000
C01080=36.365,-34.611,83.974,166.4147,-14.3117,0.0000
C01081=35.493,-35.493,84.004,166.0667,-13.9390,0.0000
C01082=34.611,-36.365,83.974,165.6883,-13.5853,0.0000
C01083=33.142,-37.858,84.019,169.0726,-15.1488,0.0000
C01084=32.045,-40.888,85.045,-179.1489,-8.2800,0.0000
C01085=34.307,-44.912,87.559,179.0888,1.2091,0.0000
C01086=38.690,-50.529,90.842,179.1404,1.1232,0.0000
C01087=44.045,-57.421,93.974,179.5702,0.5615,0.0000
C01088=9.459,-71.748,93.974,-179.9083,-0.7048,0.0000
C01089=8.371,-63.087,90.842,-179.8109,-1.3982,0.0000
C01090=7.499,-56.017,87.559,-179.7879,-1.5013,0.0000
C01091=6.253,-51.571,85.045,174.7226,6.4692,0.0000
C01092=3.334,-50.204,84.019,161.8426,3.1427,0.0000
C01093=1.241,-50.188,83.974,160.6464,-0.5465,0.0000
C01094=0.000,-50.195,84.004,160.6645,-0.0000,0.0000
C01095=0.000,-50.195,84.004,160.6645,-0.0000,0.0000
C01096=-1.240,-50.188,83.974,160.6464,0.5465,0.0000
C01097=-3.335,-50.204,84.019,161.8426,-3.1427,0.0000
C01098=-6.253,-51.571,85.045,174.7226,-6.4692,0.0000
C01099=-7.499,-56.017,87.559,-179.7879,1.5013,0.0000
C01100=-8.371,-63.087,90.842,-179.8109,1.3982,0.0000
C01101=-9.459,-71.748,93.974,-179.9083,0.7048,0.0000
C01102=-44.045,-57.421,93.974,179.5702,-0.5615,0.0000
C01103=-38.690,-50.529,90.842,179.1404,-1.1232,0.0000
C01104=-34.307,-44.912,87.559,179.0888,-1.2091,0.0000
C01105=-32.045,-40.888,85.045,-179.1489,8.2800,0.0000
C01106=-33.142,-37.857,84.019,169.0726,15.1488,0.0000
C01107=-34.611,-36.365,83.974,165.6883,13.5853,0.0000
C01108=-35.493,-35.493,84.004,166.0610,13.9333,0.0000
C01109=-36.365,-34.611,83.974,166.4147,14.3117,0.0000
C01110=-37.858,-33.142,84.019,164.8512,10.9274,0.0000
C01111=-40.888,-32.045,85.045,171.7200,-0.8511,0.0000
C01112=-44.912,-34.307,87.559,-178.7909,0.9112,0.0000
C01113=-50.529,-38.690,90.842,-178.8768,0.8596,0.0000
C01114=-57.421,-44.045,93.974,-179.4385,0.4298,0.0000
C01115=-71.748,-9.459,93.974,179.2952,-0.0917,0.0000
C01116=-63.087,-8.371,90.842,178.6018,-0.1891,0.0000
C01117=-56.017,-7.499,87.559,178.4987,-0.2121,0.0000
C01118=-51.571,-6.253,85.045,-173.5308,5.2774,0.0000
C01119=-50.204,-3.334,84.019,-176.8573,18.1574,0.0000
C01120=-50.188,-1.241,83.974,179.4535,19.3536,0.0000
C01121=-50.195,0.000,84.004,180.0000,19.3355,0.0000
C01122=-50.188,1.240,83.974,-179.4535,19.3536,0.0000
C01123=-50.204,3.335,84.019,176.8573,18.1574,0.0000
C01124=-51.571,6.253,85.045,173.5308,5.2774,0.0000
C01125=-56.017,7.499,87.559,-178.4987,-0.2121,0.0000
C01126=-63.087,8.371,90.842,-178.6018,-0.1891,0.0000
C01127=-71.748,9.459,93.974,-179.2952,-0.0917,0.0000
C01128=-57.421,44.045,93.974,179.4385,0.4298,0.0000
C01129=-50.529,38.690,90.842,178.8768,0.8596,0.0000
C01130=-44.912,34.307,87.559,178.7909,0.9112,0.0000
C01131=-40.888,32.045,85.045,-171.7200,-0.8511,0.0000
C01132=-37.857,33.142,84.019,-164.8512,10.9274,0.0000
C01133=-36.365,34.611,83.974,-166.4147,14.3117,0.0000
C01134=-35.493,35.493,84.004,-166.0667,13.9390,0.0000
C01135=-34.611,36.365,83.974,-165.6883,13.5853,0.0000
C01136=-33.142,37.858,84.019,-169.0726,15.1488,0.0000
C01137=-32.045,40.888,85.045,179.1489,8.2800,0.0000
C01138=-34.307,44.912,87.559,-179.0888,-1.2091,0.0000
C01139=-38.690,50.529,90.842,-179.1404,-1.1232,0.0000
C01140=-44.045,57.421,93.974,-179.5702,-0.5615,0.0000
C01141=-9.459,71.748,93.974,179.9083,0.7048,0.0000
C01142=-8.371,63.087,90.842,179.8109,1.3982,0.0000
C01143=-7.499,56.017,87.559,179.7879,1.5013,0.0000
C01144=-6.253,51.571,85.045,-174.7226,-6.4692,0.0000
C01145=-3.335,50.204,84.019,-161.8426,-3.1427,0.0000
C01146=-1.240,50.188,83.974,-160.6464,0.5465,0.0000
C01147=0.000,50.195,84.004,-160.6645,-0.0000,0.0000
C01148=0.000,49.517,86.097,-163.5005,-0.0000,0.0000
C01149=1.179,49.510,86.067,-163.4769,-0.4303,0.0000
C01150=3.230,49.536,86.112,-164.5754,2.7526,0.0000
C01151=6.137,50.981,87.161,-175.7730,5.2870,0.0000
C01152=7.391,55.610,89.719,179.8395,-1.1804,0.0000
C01153=8.302,62.896,93.033,179.8911,-0.8308,0.0000
C01154=38.603,50.345,93.033,-179.4900,0.6647,0.0000
C01155=34.096,44.548,89.719,-179.2780,0.9455,0.0000
C01156=31.710,40.389,87.161,179.2443,-6.7135,0.0000
C01157=32.743,37.311,86.112,-170.8506,-12.9025,0.0000
C01158=34.176,35.843,86.067,-167.8616,-11.5545,0.0000
C01159=35.014,35.014,86.097,-168.1659,-11.8284,0.0000
C01160=35.842,34.176,86.067,-168.4455,-12.1384,0.0000
C01161=37.311,32.743,86.112,-167.0975,-9.1494,0.0000
C01162=40.389,31.710,87.161,-173.2922,0.7557,0.0000
C01163=44.548,34.096,89.719,179.0545,-0.7220,0.0000
C01164=50.345,38.603,93.033,179.3353,-0.5100,0.0000
C01165=62.896,8.302,93.033,-179.1692,0.1089,0.0000
C01166=55.610,7.391,89.719,-178.8196,0.1605,0.0000
C01167=50.981,6.137,87.161,174.7130,-4.2270,0.0000
C01168=49.536,3.230,86.112,177.2474,-15.4246,0.0000
C01169=49.510,1.179,86.067,-179.5697,-16.5231,0.0000
C01170=49.517,0.000,86.097,-180.0000,-16.4995,0.0000
C01171=49.510,-1.178,86.067,179.5697,-16.5231,0.0000
C01172=49.536,-3.231,86.112,-177.2474,-15.4191,0.0000
C01173=50.981,-6.137,87.161,-174.7130,-4.2270,0.0000
C01174=55.610,-7.391,89.719,178.8196,0.1605,0.0000
C01175=62.896,-8.302,93.033,179.1692,0.1089,0.0000
C01176=50.345,-38.603,93.033,-179.3353,-0.5100,0.0000
C01177=44.548,-34.096,89.719,-179.0545,-0.7220,0.0000
C01178=40.389,-31.710,87.161,173.2865,0.7557,0.0000
C01179=37.311,-32.743,86.112,167.0975,-9.1494,0.0000
C01180=35.843,-34.176,86.067,168.4455,-12.1384,0.0000
C01181=35.014,-35.014,86.097,168.1716,-11.8341,0.0000
C01182=34.176,-35.842,86.067,167.8616,-11.5545,0.0000
C01183=32.743,-37.311,86.112,170.8506,-12.9025,0.0000
C01184=31.710,-40.389,87.161,-179.2443,-6.7078,0.0000
C01185=34.096,-44.548,89.719,179.2780,0.9455,0.0000
C01186=38.603,-50.345,93.033,179.4900,0.6647,0.0000
C01187=8.302,-62.896,93.033,-179.8911,-0.8308,0.0000
C01188=7.391,-55.610,89.719,-179.8395,-1.1804,0.0000
C01189=6.137,-50.981,87.161,175.7730,5.2870,0.0000
C01190=3.230,-49.536,86.112,164.5754,2.7526,0.0000
C01191=1.179,-49.510,86.067,163.4769,-0.4303,0.0000
C01192=0.000,-49.517,86.097,163.5005,-0.0000,0.0000
C01193=0.000,-49.517,86.097,163.5005,-0.0000,0.0000
C01194=-1.178,-49.510,86.067,163.4769,0.4303,0.0000
C01195=-3.231,-49.536,86.112,164.5809,-2.7526,0.0000
C01196=-6.137,-50.981,87.161,175.7730,-5.2870,0.0000
C01197=-7.391,-55.610,89.719,-179.8395,1.1804,0.0000
C01198=-8.302,-62.896,93.033,-179.8911,0.8308,0.0000
C01199=-38.603,-50.345,93.033,179.4900,-0.6647,0.0000
C01200=-34.096,-44.548,89.719,179.2780,-0.9455,0.0000
C01201=-31.710,-40.389,87.161,-179.2443,6.7135,0.0000
C01202=-32.743,-37.311,86.112,170.8506,12.9025,0.0000
C01203=-34.176,-35.843,86.067,167.8616,11.5545,0.0000
C01204=-35.014,-35.014,86.097,168.1659,11.8284,0.0000
C01205=-35.842,-34.176,86.067,168.4455,12.1384,0.0000
C01206=-37.311,-32.743,86.112,167.0975,9.1494,0.0000
C01207=-40.389,-31.710,87.161,173.2922,-0.7557,0.0000
C01208=-44.548,-34.096,89.719,-179.0545,0.7220,0.0000
C01209=-50.345,-38.603,93.033,-179.3353,0.5100,0.0000
C01210=-62.896,-8.302,93.033,179.1692,-0.1089,0.0000
C01211=-55.610,-7.391,89.719,178.8196,-0.1605,0.0000
C01212=-50.981,-6.137,87.161,-174.7130,4.2270,0.0000
C01213=-49.536,-3.230,86.112,-177.2474,15.4246,0.0000
C01214=-49.510,-1.179,86.067,179.5697,16.5231,0.0000
C01215=-49.517,0.000,86.097,180.0000,16.4995,0.0000
C01216=-49.510,1.178,86.067,-179.5697,16.5231,0.0000
C01217=-49.536,3.231,86.112,177.2474,15.4191,0.0000
C01218=-50.981,6.137,87.161,174.7130,4.2270,0.0000
C01219=-55.610,7.391,89.719,-178.8196,-0.1605,0.0000
C01220=-62.896,8.302,93.033,-179.1692,-0.1089,0.0000
C01221=-50.345,38.603,93.033,179.3353,0.5100,0.0000
C01222=-44.548,34.096,89.719,179.0545,0.7220,0.0000
C01223=-40.389,31.710,87.161,-173.2865,-0.7557,0.0000
C01224=-37.311,32.743,86.112,-167.0975,9.1494,0.0000
C01225=-35.843,34.176,86.067,-168.4455,12.1384,0.0000
C01226=-35.014,35.014,86.097,-168.1716,11.8341,0.0000
C01227=-34.176,35.842,86.067,-167.8616,11.5545,0.0000
C01228=-32.743,37.311,86.112,-170.8506,12.9025,0.0000
C01229=-31.710,40.389,87.161,179.2443,6.7078,0.0000
C01230=-34.096,44.548,89.719,-179.2780,-0.9455,0.0000
C01231=-38.603,50.345,93.033,-179.4900,-0.6647,0.0000
C01232=-8.302,62.896,93.033,179.8911,0.8308,0.0000
C01233=-7.391,55.610,89.719,179.8395,1.1804,0.0000
C01234=-6.137,50.981,87.161,-175.7730,-5.2870,0.0000
C01235=-3.231,49.536,86.112,-164.5809,-2.7526,0.0000
C01236=-1.178,49.510,86.067,-163.4769,0.4303,0.0000
C01237=0.000,49.517,86.097,-163.5005,-0.0000,0.0000
C01238=0.000,48.949,88.223,-166.6210,-0.0000,0.0000
C01239=1.127,48.942,88.191,-166.5905,-0.3240,0.0000
C01240=3.143,48.975,88.238,-167.5520,2.2770,0.0000
C01241=6.042,50.501,89.306,-176.8106,4.0603,0.0000
C01242=7.312,55.314,91.898,179.8911,-0.8022,0.0000
C01243=8.270,62.805,95.231,179.9714,-0.2177,0.0000
C01244=38.562,50.258,95.231,-179.8625,0.1776,0.0000
C01245=33.942,44.284,91.898,-179.5072,0.6418,0.0000
C01246=31.437,39.982,89.306,179.3845,-5.1234,0.0000
C01247=32.408,36.853,88.238,-172.7059,-10.4345,0.0000
C01248=33.811,35.404,88.191,-170.2123,-9.3467,0.0000
C01249=34.612,34.612,88.223,-170.4546,-9.5454,0.0000
C01250=35.404,33.811,88.191,-170.6533,-9.7877,0.0000
C01251=36.854,32.408,88.238,-169.5655,-7.2941,0.0000
C01252=39.982,31.437,89.306,-174.8823,0.6155,0.0000
C01253=44.284,33.942,91.898,179.3582,-0.4928,0.0000
C01254=50.258,38.562,95.231,179.8224,-0.1375,0.0000
C01255=62.805,8.270,95.231,-179.7823,0.0286,0.0000
C01256=55.314,7.312,91.898,-179.1978,0.1089,0.0000
C01257=50.501,6.042,89.306,175.9397,-3.1894,0.0000
C01258=48.975,3.143,88.238,177.7230,-12.4480,0.0000
C01259=48.942,1.127,88.191,-179.6760,-13.4095,0.0000
C01260=48.949,0.000,88.223,-180.0000,-13.3790,0.0000
C01261=48.942,-1.126,88.191,179.6760,-13.4095,0.0000
C01262=48.976,-3.143,88.238,-177.7230,-12.4480,0.0000
C01263=50.501,-6.042,89.306,-175.9397,-3.1894,0.0000
C01264=55.314,-7.312,91.898,179.1978,0.1089,0.0000
C01265=62.805,-8.270,95.231,179.7823,0.0286,0.0000
C01266=50.258,-38.562,95.231,-179.8224,-0.1375,0.0000
C01267=44.284,-33.942,91.898,-179.3582,-0.4928,0.0000
C01268=39.982,-31.437,89.306,174.8766,0.6155,0.0000
C01269=36.853,-32.408,88.238,169.5655,-7.2941,0.0000
C01270=35.404,-33.811,88.191,170.6533,-9.7877,0.0000
C01271=34.612,-34.612,88.223,170.4546,-9.5454,0.0000
C01272=33.811,-35.404,88.191,170.2123,-9.3467,0.0000
C01273=32.408,-36.854,88.238,172.7059,-10.4345,0.0000
C01274=31.437,-39.982,89.306,-179.3845,-5.1177,0.0000
C01275=33.942,-44.284,91.898,179.5072,0.6418,0.0000
C01276=38.562,-50.258,95.231,179.8625,0.1776,0.0000
C01277=8.270,-62.805,95.231,-179.9714,-0.2177,0.0000
C01278=7.312,-55.314,91.898,-179.8911,-0.8022,0.0000
C01279=6.042,-50.501,89.306,176.8106,4.0603,0.0000
C01280=3.143,-48.975,88.238,167.5520,2.2770,0.0000
C01281=1.127,-48.942,88.191,166.5905,-0.3240,0.0000
C01282=0.000,-48.949,88.223,166.6210,-0.0000,0.0000
C01283=0.000,-48.949,88.223,166.6210,-0.0000,0.0000
C01284=-1.126,-48.942,88.191,166.5905,0.3240,0.0000
C01285=-3.143,-48.976,88.238,167.5520,-2.2770,0.0000
C01286=-6.042,-50.501,89.306,176.8106,-4.0603,0.0000
C01287=-7.312,-55.314,91.898,-179.8911,0.8022,0.0000
C01288=-8.270,-62.805,95.231,-179.9714,0.2177,0.0000
C01289=-38.562,-50.258,95.231,179.8625,-0.1776,0.0000
C01290=-33.942,-44.284,91.898,179.5072,-0.6418,0.0000
C01291=-31.437,-39.982,89.306,-179.3845,5.1234,0.0000
C01292=-32.408,-36.853,88.238,172.7059,10.4345,0.0000
C01293=-33.811,-35.404,88.191,170.2123,9.3467,0.0000
C01294=-34.612,-34.612,88.223,170.4546,9.5454,0.0000
C01295=-35.404,-33.811,88.191,170.6533,9.7877,0.0000
C01296=-36.854,-32.408,88.238,169.5655,7.2941,0.0000
C01297=-39.982,-31.437,89.306,174.8823,-0.6155,0.0000
C01298=-44.284,-33.942,91.898,-179.3582,0.4928,0.0000
C01299=-50.258,-38.562,95.231,-179.8224,0.1375,0.0000
C01300=-62.805,-8.270,95.231,179.7823,-0.0286,0.0000
C01301=-55.314,-7.312,91.898,179.1978,-0.1089,0.0000
C01302=-50.501,-6.042,89.306,-175.9397,3.1894,0.0000
C01303=-48.975,-3.143,88.238,-177.7230,12.4480,0.0000
C01304=-48.942,-1.127,88.191,179.6760,13.4095,0.0000
C01305=-48.949,0.000,88.223,180.0000,13.3790,0.0000
C01306=-48.942,1.126,88.191,-179.6760,13.4095,0.0000
C01307=-48.976,3.143,88.238,177.7230,12.4480,0.0000
C01308=-50.501,6.042,89.306,175.9397,3.1894,0.0000
C01309=-55.314,7.312,91.898,-179.1978,-0.1089,0.0000
C01310=-62.805,8.270,95.231,-179.7823,-0.0286,0.0000
C01311=-50.258,38.562,95.231,179.8224,0.1375,0.0000
C01312=-44.284,33.942,91.898,179.3582,0.4928,0.0000
C01313=-39.982,31.437,89.306,-174.8766,-0.6155,0.0000
C01314=-36.853,32.408,88.238,-169.5655,7.2941,0.0000
C01315=-35.404,33.811,88.191,-170.6533,9.7877,0.0000
C01316=-34.612,34.612,88.223,-170.4546,9.5454,0.0000
C01317=-33.811,35.404,88.191,-170.2123,9.3467,0.0000
C01318=-32.408,36.854,88.238,-172.7059,10.4345,0.0000
C01319=-31.437,39.982,89.306,179.3845,5.1177,0.0000
C01320=-33.942,44.284,91.898,-179.5072,-0.6418,0.0000
C01321=-38.562,50.258,95.231,-179.8625,-0.1776,0.0000
C01322=-8.270,62.805,95.231,179.9714,0.2177,0.0000
C01323=-7.312,55.314,91.898,179.8911,0.8022,0.0000
C01324=-6.042,50.501,89.306,-176.8106,-4.0603,0.0000
C01325=-3.143,48.976,88.238,-167.5520,-2.2770,0.0000
C01326=-1.126,48.942,88.191,-166.5905,0.3240,0.0000
C01327=0.000,48.949,88.223,-166.6210,-0.0000,0.0000
C01328=0.000,48.503,90.377,-170.0375,-0.0000,0.0000
C01329=1.086,48.496,90.345,-169.9970,-0.2269,0.0000
C01330=3.075,48.536,90.393,-170.7657,1.7185,0.0000
C01331=5.972,50.143,91.476,-177.8369,2.7877,0.0000
C01332=7.266,55.138,94.090,179.9484,-0.3896,0.0000
C01333=33.851,44.126,94.090,-179.7651,0.3094,0.0000
C01334=31.234,39.679,91.476,179.5580,-3.4973,0.0000
C01335=32.146,36.494,90.393,-174.6438,-7.7517,0.0000
C01336=33.524,35.059,90.345,-172.7375,-6.9531,0.0000
C01337=34.297,34.297,90.377,-172.9158,-7.0842,0.0000
C01338=35.059,33.525,90.345,-173.0469,-7.2625,0.0000
C01339=36.495,32.146,90.393,-172.2483,-5.3504,0.0000
C01340=39.679,31.234,91.476,-176.5027,0.4420,0.0000
C01341=44.126,33.851,94.090,179.6906,-0.2349,0.0000
C01342=55.138,7.266,94.090,-179.6104,0.0516,0.0000
C01343=50.143,5.972,91.476,177.2123,-2.1631,0.0000
C01344=48.536,3.075,90.393,178.2815,-9.2343,0.0000
C01345=48.496,1.086,90.345,-179.7731,-10.0030,0.0000
C01346=48.503,0.000,90.377,-180.0000,-9.9625,0.0000
C01347=48.496,-1.085,90.345,179.7731,-10.0030,0.0000
C01348=48.536,-3.075,90.393,-178.2815,-9.2343,0.0000
C01349=50.143,-5.972,91.476,-177.2123,-2.1631,0.0000
C01350=55.138,-7.266,94.090,179.6104,0.0516,0.0000
C01351=44.126,-33.851,94.090,-179.6906,-0.2349,0.0000
C01352=39.679,-31.234,91.476,176.5027,0.4420,0.0000
C01353=36.494,-32.146,90.393,172.2483,-5.3562,0.0000
C01354=35.059,-33.524,90.345,173.0469,-7.2625,0.0000
C01355=34.297,-34.297,90.377,172.9158,-7.0842,0.0000
C01356=33.525,-35.059,90.345,172.7375,-6.9531,0.0000
C01357=32.146,-36.495,90.393,174.6496,-7.7517,0.0000
C01358=31.234,-39.679,91.476,-179.5580,-3.4973,0.0000
C01359=33.851,-44.126,94.090,179.7651,0.3094,0.0000
C01360=7.266,-55.138,94.090,-179.9484,-0.3896,0.0000
C01361=5.972,-50.143,91.476,177.8369,2.7877,0.0000
C01362=3.075,-48.536,90.393,170.7657,1.7185,0.0000
C01363=1.086,-48.496,90.345,169.9970,-0.2269,0.0000
C01364=0.000,-48.503,90.377,170.0375,-0.0000,0.0000
C01365=0.000,-48.503,90.377,170.0375,-0.0000,0.0000
C01366=-1.085,-48.496,90.345,169.9970,0.2269,0.0000
C01367=-3.075,-48.536,90.393,170.7657,-1.7185,0.0000
C01368=-5.972,-50.143,91.476,177.8369,-2.7877,0.0000
C01369=-7.266,-55.138,94.090,-179.9484,0.3896,0.0000
C01370=-33.851,-44.126,94.090,179.7651,-0.3094,0.0000
C01371=-31.234,-39.679,91.476,-179.5580,3.4973,0.0000
C01372=-32.146,-36.494,90.393,174.6438,7.7517,0.0000
C01373=-33.524,-35.059,90.345,172.7375,6.9531,0.0000
C01374=-34.297,-34.297,90.377,172.9158,7.0842,0.0000
C01375=-35.059,-33.525,90.345,173.0469,7.2625,0.0000
C01376=-36.495,-32.146,90.393,172.2483,5.3504,0.0000
C01377=-39.679,-31.234,91.476,176.5027,-0.4420,0.0000
C01378=-44.126,-33.851,94.090,-179.6906,0.2349,0.0000
C01379=-55.138,-7.266,94.090,179.6104,-0.0516,0.0000
C01380=-50.143,-5.972,91.476,-177.2123,2.1631,0.0000
C01381=-48.536,-3.075,90.393,-178.2815,9.2343,0.0000
C01382=-48.496,-1.086,90.345,179.7731,10.0030,0.0000
C01383=-48.503,0.000,90.377,180.0000,9.9625,0.0000
C01384=-48.496,1.085,90.345,-179.7731,10.0030,0.0000
C01385=-48.536,3.075,90.393,178.2815,9.2343,0.0000
C01386=-50.143,5.972,91.476,177.2123,2.1631,0.0000
C01387=-55.138,7.266,94.090,-179.6104,-0.0516,0.0000
C01388=-44.126,33.851,94.090,179.6906,0.2349,0.0000
C01389=-39.679,31.234,91.476,-176.5027,-0.4420,0.0000
C01390=-36.494,32.146,90.393,-172.2483,5.3562,0.0000
C01391=-35.059,33.524,90.345,-173.0469,7.2625,0.0000
C01392=-34.297,34.297,90.377,-172.9158,7.0842,0.0000
C01393=-33.525,35.059,90.345,-172.7375,6.9531,0.0000
C01394=-32.146,36.495,90.393,-174.6496,7.7517,0.0000
C01395=-31.234,39.679,91.476,179.5580,3.4973,0.0000
C01396=-33.851,44.126,94.090,-179.7651,-0.3094,0.0000
C01397=-7.266,55.138,94.090,179.9484,0.3896,0.0000
C01398=-5.972,50.143,91.476,-177.8369,-2.7877,0.0000
C01399=-3.075,48.536,90.393,-170.7657,-1.7185,0.0000
C01400=-1.085,48.496,90.345,-169.9970,0.2269,0.0000
C01401=0.000,48.503,90.377,-170.0375,-0.0000,0.0000
C01402=0.000,48.191,92.555,-173.7250,-0.0000,0.0000
C01403=1.057,48.183,92.523,-173.6788,-0.1326,0.0000
C01404=3.027,48.229,92.571,-174.2136,1.0885,0.0000
C01405=5.927,49.917,93.664,-178.8709,1.4615,0.0000
C01406=31.106,39.488,93.664,179.7650,-1.8338,0.0000
C01407=31.963,36.244,92.571,-176.6687,-4.8671,0.0000
C01408=33.323,34.818,92.523,-175.4268,-4.3842,0.0000
C01409=34.076,34.076,92.555,-175.5533,-4.4467,0.0000
C01410=34.818,33.324,92.523,-175.6158,-4.5732,0.0000
C01411=36.244,31.963,92.571,-175.1329,-3.3313,0.0000
C01412=39.488,31.106,93.664,-178.1662,0.2350,0.0000
C01413=49.917,5.927,93.664,178.5385,-1.1291,0.0000
C01414=48.229,3.027,92.571,178.9115,-5.7864,0.0000
C01415=48.183,1.057,92.523,-179.8674,-6.3212,0.0000
C01416=48.191,0.000,92.555,-180.0000,-6.2750,0.0000
C01417=48.183,-1.057,92.523,179.8674,-6.3212,0.0000
C01418=48.229,-3.027,92.571,-178.9057,-5.7864,0.0000
C01419=49.918,-5.927,93.664,-178.5385,-1.1291,0.0000
C01420=39.488,-31.106,93.664,178.1662,0.2350,0.0000
C01421=36.244,-31.963,92.571,175.1329,-3.3313,0.0000
C01422=34.818,-33.323,92.523,175.6158,-4.5732,0.0000
C01423=34.076,-34.076,92.555,175.5533,-4.4467,0.0000
C01424=33.324,-34.818,92.523,175.4268,-4.3842,0.0000
C01425=31.963,-36.244,92.571,176.6687,-4.8671,0.0000
C01426=31.106,-39.488,93.664,-179.7650,-1.8338,0.0000
C01427=5.927,-49.917,93.664,178.8709,1.4615,0.0000
C01428=3.027,-48.229,92.571,174.2136,1.0885,0.0000
C01429=1.057,-48.183,92.523,173.6788,-0.1326,0.0000
C01430=0.000,-48.191,92.555,173.7250,-0.0000,0.0000
C01431=0.000,-48.191,92.555,173.7250,-0.0000,0.0000
C01432=-1.057,-48.183,92.523,173.6788,0.1326,0.0000
C01433=-3.027,-48.229,92.571,174.2136,-1.0943,0.0000
C01434=-5.927,-49.918,93.664,178.8709,-1.4615,0.0000
C01435=-31.106,-39.488,93.664,-179.7650,1.8338,0.0000
C01436=-31.963,-36.244,92.571,176.6687,4.8671,0.0000
C01437=-33.323,-34.818,92.523,175.4268,4.3842,0.0000
C01438=-34.076,-34.076,92.555,175.5533,4.4467,0.0000
C01439=-34.818,-33.324,92.523,175.6158,4.5732,0.0000
C01440=-36.244,-31.963,92.571,175.1329,3.3313,0.0000
C01441=-39.488,-31.106,93.664,178.1662,-0.2350,0.0000
C01442=-49.917,-5.927,93.664,-178.5385,1.1291,0.0000
C01443=-48.229,-3.027,92.571,-178.9115,5.7864,0.0000
C01444=-48.183,-1.057,92.523,179.8674,6.3212,0.0000
C01445=-48.191,0.000,92.555,180.0000,6.2750,0.0000
C01446=-48.183,1.057,92.523,-179.8674,6.3212,0.0000
C01447=-48.229,3.027,92.571,178.9057,5.7864,0.0000
C01448=-49.918,5.927,93.664,178.5385,1.1291,0.0000
C01449=-39.488,31.106,93.664,-178.1662,-0.2350,0.0000
C01450=-36.244,31.963,92.571,-175.1329,3.3313,0.0000
C01451=-34.818,33.323,92.523,-175.6158,4.5732,0.0000
C01452=-34.076,34.076,92.555,-175.5533,4.4467,0.0000
C01453=-33.324,34.818,92.523,-175.4268,4.3842,0.0000
C01454=-31.963,36.244,92.571,-176.6687,4.8671,0.0000
C01455=-31.106,39.488,93.664,179.7650,1.8338,0.0000
C01456=-5.927,49.918,93.664,-178.8709,-1.4615,0.0000
C01457=-3.027,48.229,92.571,-174.2136,-1.0943,0.0000
C01458=-1.057,48.183,92.523,-173.6788,0.1326,0.0000
C01459=0.000,48.191,92.555,-173.7250,-0.0000,0.0000
C01460=0.000,48.026,94.749,-177.6675,-0.0000,0.0000
C01461=1.042,48.016,94.716,-177.6100,-0.0516,0.0000
C01462=3.002,48.067,94.764,-177.8681,0.4071,0.0000
C01463=5.911,49.834,95.862,-179.9312,0.0859,0.0000
C01464=31.058,39.418,95.862,179.9828,-0.1089,0.0000
C01465=31.866,36.111,94.764,-178.7789,-1.7940,0.0000
C01466=33.216,34.689,94.716,-178.2744,-1.6569,0.0000
C01467=33.959,33.959,94.749,-178.3490,-1.6510,0.0000
C01468=34.689,33.216,94.716,-178.3431,-1.7256,0.0000
C01469=36.111,31.865,94.764,-178.2060,-1.2211,0.0000
C01470=39.418,31.058,95.862,-179.8911,0.0172,0.0000
C01471=49.834,5.911,95.862,179.9141,-0.0688,0.0000
C01472=48.067,3.002,94.764,179.5929,-2.1319,0.0000
C01473=48.016,1.042,94.716,-179.9484,-2.3900,0.0000
C01474=48.026,0.000,94.749,-180.0000,-2.3325,0.0000
C01475=48.016,-1.041,94.716,179.9484,-2.3900,0.0000
C01476=48.067,-3.002,94.764,-179.5929,-2.1319,0.0000
C01477=49.834,-5.911,95.862,-179.9141,-0.0688,0.0000
C01478=39.418,-31.058,95.862,179.8911,0.0172,0.0000
C01479=36.111,-31.866,94.764,178.2060,-1.2211,0.0000
C01480=34.689,-33.216,94.716,178.3431,-1.7256,0.0000
C01481=33.959,-33.959,94.749,178.3490,-1.6510,0.0000
C01482=33.216,-34.689,94.716,178.2744,-1.6569,0.0000
C01483=31.865,-36.111,94.764,178.7789,-1.7940,0.0000
C01484=31.058,-39.418,95.862,-179.9828,-0.1089,0.0000
C01485=5.911,-49.834,95.862,179.9312,0.0859,0.0000
C01486=3.002,-48.067,94.764,177.8681,0.4071,0.0000
C01487=1.042,-48.016,94.716,177.6100,-0.0516,0.0000
C01488=0.000,-48.026,94.749,177.6675,-0.0000,0.0000
C01489=0.000,-48.026,94.749,177.6675,-0.0000,0.0000
C01490=-1.041,-48.016,94.716,177.6100,0.0516,0.0000
C01491=-3.002,-48.067,94.764,177.8681,-0.4071,0.0000
C01492=-5.911,-49.834,95.862,179.9312,-0.0859,0.0000
C01493=-31.058,-39.418,95.862,-179.9828,0.1089,0.0000
C01494=-31.866,-36.111,94.764,178.7789,1.7940,0.0000
C01495=-33.216,-34.689,94.716,178.2744,1.6569,0.0000
C01496=-33.959,-33.959,94.749,178.3490,1.6510,0.0000
C01497=-34.689,-33.216,94.716,178.3431,1.7256,0.0000
C01498=-36.111,-31.865,94.764,178.2060,1.2211,0.0000
C01499=-39.418,-31.058,95.862,179.8911,-0.0172,0.0000
C01500=-49.834,-5.911,95.862,-179.9141,0.0688,0.0000
C01501=-48.067,-3.002,94.764,-179.5929,2.1319,0.0000
C01502=-48.016,-1.042,94.716,179.9484,2.3900,0.0000
C01503=-48.026,0.000,94.749,180.0000,2.3325,0.0000
C01504=-48.016,1.041,94.716,-179.9484,2.3900,0.0000
C01505=-48.067,3.002,94.764,179.5929,2.1319,0.0000
C01506=-49.834,5.911,95.862,179.9141,0.0688,0.0000
C01507=-39.418,31.058,95.862,-179.8911,-0.0172,0.0000
C01508=-36.111,31.866,94.764,-178.2060,1.2211,0.0000
C01509=-34.689,33.216,94.716,-178.3431,1.7256,0.0000
C01510=-33.959,33.959,94.749,-178.3490,1.6510,0.0000
C01511=-33.216,34.689,94.716,-178.2744,1.6569,0.0000
C01512=-31.865,36.111,94.764,-178.7789,1.7940,0.0000
C01513=-31.058,39.418,95.862,179.9828,0.1089,0.0000
C01514=-5.911,49.834,95.862,-179.9312,-0.0859,0.0000
C01515=-3.002,48.067,94.764,-177.8681,-0.4071,0.0000
C01516=-1.041,48.016,94.716,-177.6100,0.0516,0.0000
C01517=0.000,48.026,94.749,-177.6675,-0.0000,0.0000
//INST
<<<<<<< HEAD
///DATE 2022/04/08 11:22
=======
///DATE 2022/04/07 19:01
>>>>>>> 4879be8d801170d946a7a1e3411c19a4bc0e02c8
///COMM
///ATTR SC,RW,RJ
////FRAME USER 2
///GROUP1 RB1
NOP
MOVL C00000
MOVL C00001
MOVL C00002
MOVL C00003
MOVL C00004
MOVL C00005
MOVL C00006
MOVL C00007
MOVL C00008
MOVL C00009
MOVL C00010
MOVL C00011
MOVL C00012
MOVL C00013
MOVL C00014
MOVL C00015
MOVL C00016
MOVL C00017
MOVL C00018
MOVL C00019
MOVL C00020
MOVL C00021
MOVL C00022
MOVL C00023
MOVL C00024
MOVL C00025
MOVL C00026
MOVL C00027
MOVL C00028
MOVL C00029
MOVL C00030
MOVL C00031
MOVL C00032
MOVL C00033
MOVL C00034
MOVL C00035
MOVL C00036
MOVL C00037
MOVL C00038
MOVL C00039
MOVL C00040
MOVL C00041
MOVL C00042
MOVL C00043
MOVL C00044
MOVL C00045
MOVL C00046
MOVL C00047
MOVL C00048
MOVL C00049
MOVL C00050
MOVL C00051
MOVL C00052
MOVL C00053
MOVL C00054
MOVL C00055
MOVL C00056
MOVL C00057
MOVL C00058
MOVL C00059
MOVL C00060
MOVL C00061
MOVL C00062
MOVL C00063
MOVL C00064
MOVL C00065
MOVL C00066
MOVL C00067
MOVL C00068
MOVL C00069
MOVL C00070
MOVL C00071
MOVL C00072
MOVL C00073
MOVL C00074
MOVL C00075
MOVL C00076
MOVL C00077
MOVL C00078
MOVL C00079
MOVL C00080
MOVL C00081
MOVL C00082
MOVL C00083
MOVL C00084
MOVL C00085
MOVL C00086
MOVL C00087
MOVL C00088
MOVL C00089
MOVL C00090
MOVL C00091
MOVL C00092
MOVL C00093
MOVL C00094
MOVL C00095
MOVL C00096
MOVL C00097
MOVL C00098
MOVL C00099
MOVL C00100
MOVL C00101
MOVL C00102
MOVL C00103
MOVL C00104
MOVL C00105
MOVL C00106
MOVL C00107
MOVL C00108
MOVL C00109
MOVL C00110
MOVL C00111
MOVL C00112
MOVL C00113
MOVL C00114
MOVL C00115
MOVL C00116
MOVL C00117
MOVL C00118
MOVL C00119
MOVL C00120
MOVL C00121
MOVL C00122
MOVL C00123
MOVL C00124
MOVL C00125
MOVL C00126
MOVL C00127
MOVL C00128
MOVL C00129
MOVL C00130
MOVL C00131
MOVL C00132
MOVL C00133
MOVL C00134
MOVL C00135
MOVL C00136
MOVL C00137
MOVL C00138
MOVL C00139
MOVL C00140
MOVL C00141
MOVL C00142
MOVL C00143
MOVL C00144
MOVL C00145
MOVL C00146
MOVL C00147
MOVL C00148
MOVL C00149
MOVL C00150
MOVL C00151
MOVL C00152
MOVL C00153
MOVL C00154
MOVL C00155
MOVL C00156
MOVL C00157
MOVL C00158
MOVL C00159
MOVL C00160
MOVL C00161
MOVL C00162
MOVL C00163
MOVL C00164
MOVL C00165
MOVL C00166
MOVL C00167
MOVL C00168
MOVL C00169
MOVL C00170
MOVL C00171
MOVL C00172
MOVL C00173
MOVL C00174
MOVL C00175
MOVL C00176
MOVL C00177
MOVL C00178
MOVL C00179
MOVL C00180
MOVL C00181
MOVL C00182
MOVL C00183
MOVL C00184
MOVL C00185
MOVL C00186
MOVL C00187
MOVL C00188
MOVL C00189
MOVL C00190
MOVL C00191
MOVL C00192
MOVL C00193
MOVL C00194
MOVL C00195
MOVL C00196
MOVL C00197
MOVL C00198
MOVL C00199
MOVL C00200
MOVL C00201
MOVL C00202
MOVL C00203
MOVL C00204
MOVL C00205
MOVL C00206
MOVL C00207
MOVL C00208
MOVL C00209
MOVL C00210
MOVL C00211
MOVL C00212
MOVL C00213
MOVL C00214
MOVL C00215
MOVL C00216
MOVL C00217
MOVL C00218
MOVL C00219
MOVL C00220
MOVL C00221
MOVL C00222
MOVL C00223
MOVL C00224
MOVL C00225
MOVL C00226
MOVL C00227
MOVL C00228
MOVL C00229
MOVL C00230
MOVL C00231
MOVL C00232
MOVL C00233
MOVL C00234
MOVL C00235
MOVL C00236
MOVL C00237
MOVL C00238
MOVL C00239
MOVL C00240
MOVL C00241
MOVL C00242
MOVL C00243
MOVL C00244
MOVL C00245
MOVL C00246
MOVL C00247
MOVL C00248
MOVL C00249
MOVL C00250
MOVL C00251
MOVL C00252
MOVL C00253
MOVL C00254
MOVL C00255
MOVL C00256
MOVL C00257
MOVL C00258
MOVL C00259
MOVL C00260
MOVL C00261
MOVL C00262
MOVL C00263
MOVL C00264
MOVL C00265
MOVL C00266
MOVL C00267
MOVL C00268
MOVL C00269
MOVL C00270
MOVL C00271
MOVL C00272
MOVL C00273
MOVL C00274
MOVL C00275
MOVL C00276
MOVL C00277
MOVL C00278
MOVL C00279
MOVL C00280
MOVL C00281
MOVL C00282
MOVL C00283
MOVL C00284
MOVL C00285
MOVL C00286
MOVL C00287
MOVL C00288
MOVL C00289
MOVL C00290
MOVL C00291
MOVL C00292
MOVL C00293
MOVL C00294
MOVL C00295
MOVL C00296
MOVL C00297
MOVL C00298
MOVL C00299
MOVL C00300
MOVL C00301
MOVL C00302
MOVL C00303
MOVL C00304
MOVL C00305
MOVL C00306
MOVL C00307
MOVL C00308
MOVL C00309
MOVL C00310
MOVL C00311
MOVL C00312
MOVL C00313
MOVL C00314
MOVL C00315
MOVL C00316
MOVL C00317
MOVL C00318
MOVL C00319
MOVL C00320
MOVL C00321
MOVL C00322
MOVL C00323
MOVL C00324
MOVL C00325
MOVL C00326
MOVL C00327
MOVL C00328
MOVL C00329
MOVL C00330
MOVL C00331
MOVL C00332
MOVL C00333
MOVL C00334
MOVL C00335
MOVL C00336
MOVL C00337
MOVL C00338
MOVL C00339
MOVL C00340
MOVL C00341
MOVL C00342
MOVL C00343
MOVL C00344
MOVL C00345
MOVL C00346
MOVL C00347
MOVL C00348
MOVL C00349
MOVL C00350
MOVL C00351
MOVL C00352
MOVL C00353
MOVL C00354
MOVL C00355
MOVL C00356
MOVL C00357
MOVL C00358
MOVL C00359
MOVL C00360
MOVL C00361
MOVL C00362
MOVL C00363
MOVL C00364
MOVL C00365
MOVL C00366
MOVL C00367
MOVL C00368
MOVL C00369
MOVL C00370
MOVL C00371
MOVL C00372
MOVL C00373
MOVL C00374
MOVL C00375
MOVL C00376
MOVL C00377
MOVL C00378
MOVL C00379
MOVL C00380
MOVL C00381
MOVL C00382
MOVL C00383
MOVL C00384
MOVL C00385
MOVL C00386
MOVL C00387
MOVL C00388
MOVL C00389
MOVL C00390
MOVL C00391
MOVL C00392
MOVL C00393
MOVL C00394
MOVL C00395
MOVL C00396
MOVL C00397
MOVL C00398
MOVL C00399
MOVL C00400
MOVL C00401
MOVL C00402
MOVL C00403
MOVL C00404
MOVL C00405
MOVL C00406
MOVL C00407
MOVL C00408
MOVL C00409
MOVL C00410
MOVL C00411
MOVL C00412
MOVL C00413
MOVL C00414
MOVL C00415
MOVL C00416
MOVL C00417
MOVL C00418
MOVL C00419
MOVL C00420
MOVL C00421
MOVL C00422
MOVL C00423
MOVL C00424
MOVL C00425
MOVL C00426
MOVL C00427
MOVL C00428
MOVL C00429
MOVL C00430
MOVL C00431
MOVL C00432
MOVL C00433
MOVL C00434
MOVL C00435
MOVL C00436
MOVL C00437
MOVL C00438
MOVL C00439
MOVL C00440
MOVL C00441
MOVL C00442
MOVL C00443
MOVL C00444
MOVL C00445
MOVL C00446
MOVL C00447
MOVL C00448
MOVL C00449
MOVL C00450
MOVL C00451
MOVL C00452
MOVL C00453
MOVL C00454
MOVL C00455
MOVL C00456
MOVL C00457
MOVL C00458
MOVL C00459
MOVL C00460
MOVL C00461
MOVL C00462
MOVL C00463
MOVL C00464
MOVL C00465
MOVL C00466
MOVL C00467
MOVL C00468
MOVL C00469
MOVL C00470
MOVL C00471
MOVL C00472
MOVL C00473
MOVL C00474
MOVL C00475
MOVL C00476
MOVL C00477
MOVL C00478
MOVL C00479
MOVL C00480
MOVL C00481
MOVL C00482
MOVL C00483
MOVL C00484
MOVL C00485
MOVL C00486
MOVL C00487
MOVL C00488
MOVL C00489
MOVL C00490
MOVL C00491
MOVL C00492
MOVL C00493
MOVL C00494
MOVL C00495
MOVL C00496
MOVL C00497
MOVL C00498
MOVL C00499
MOVL C00500
MOVL C00501
MOVL C00502
MOVL C00503
MOVL C00504
MOVL C00505
MOVL C00506
MOVL C00507
MOVL C00508
MOVL C00509
MOVL C00510
MOVL C00511
MOVL C00512
MOVL C00513
MOVL C00514
MOVL C00515
MOVL C00516
MOVL C00517
MOVL C00518
MOVL C00519
MOVL C00520
MOVL C00521
MOVL C00522
MOVL C00523
MOVL C00524
MOVL C00525
MOVL C00526
MOVL C00527
MOVL C00528
MOVL C00529
MOVL C00530
MOVL C00531
MOVL C00532
MOVL C00533
MOVL C00534
MOVL C00535
MOVL C00536
MOVL C00537
MOVL C00538
MOVL C00539
MOVL C00540
MOVL C00541
MOVL C00542
MOVL C00543
MOVL C00544
MOVL C00545
MOVL C00546
MOVL C00547
MOVL C00548
MOVL C00549
MOVL C00550
MOVL C00551
MOVL C00552
MOVL C00553
MOVL C00554
MOVL C00555
MOVL C00556
MOVL C00557
MOVL C00558
MOVL C00559
MOVL C00560
MOVL C00561
MOVL C00562
MOVL C00563
MOVL C00564
MOVL C00565
MOVL C00566
MOVL C00567
MOVL C00568
MOVL C00569
MOVL C00570
MOVL C00571
MOVL C00572
MOVL C00573
MOVL C00574
MOVL C00575
MOVL C00576
MOVL C00577
MOVL C00578
MOVL C00579
MOVL C00580
MOVL C00581
MOVL C00582
MOVL C00583
MOVL C00584
MOVL C00585
MOVL C00586
MOVL C00587
MOVL C00588
MOVL C00589
MOVL C00590
MOVL C00591
MOVL C00592
MOVL C00593
MOVL C00594
MOVL C00595
MOVL C00596
MOVL C00597
MOVL C00598
MOVL C00599
MOVL C00600
MOVL C00601
MOVL C00602
MOVL C00603
MOVL C00604
MOVL C00605
MOVL C00606
MOVL C00607
MOVL C00608
MOVL C00609
MOVL C00610
MOVL C00611
MOVL C00612
MOVL C00613
MOVL C00614
MOVL C00615
MOVL C00616
MOVL C00617
MOVL C00618
MOVL C00619
MOVL C00620
MOVL C00621
MOVL C00622
MOVL C00623
MOVL C00624
MOVL C00625
MOVL C00626
MOVL C00627
MOVL C00628
MOVL C00629
MOVL C00630
MOVL C00631
MOVL C00632
MOVL C00633
MOVL C00634
MOVL C00635
MOVL C00636
MOVL C00637
MOVL C00638
MOVL C00639
MOVL C00640
MOVL C00641
MOVL C00642
MOVL C00643
MOVL C00644
MOVL C00645
MOVL C00646
MOVL C00647
MOVL C00648
MOVL C00649
MOVL C00650
MOVL C00651
MOVL C00652
MOVL C00653
MOVL C00654
MOVL C00655
MOVL C00656
MOVL C00657
MOVL C00658
MOVL C00659
MOVL C00660
MOVL C00661
MOVL C00662
MOVL C00663
MOVL C00664
MOVL C00665
MOVL C00666
MOVL C00667
MOVL C00668
MOVL C00669
MOVL C00670
MOVL C00671
MOVL C00672
MOVL C00673
MOVL C00674
MOVL C00675
MOVL C00676
MOVL C00677
MOVL C00678
MOVL C00679
MOVL C00680
MOVL C00681
MOVL C00682
MOVL C00683
MOVL C00684
MOVL C00685
MOVL C00686
MOVL C00687
MOVL C00688
MOVL C00689
MOVL C00690
MOVL C00691
MOVL C00692
MOVL C00693
MOVL C00694
MOVL C00695
MOVL C00696
MOVL C00697
MOVL C00698
MOVL C00699
MOVL C00700
MOVL C00701
MOVL C00702
MOVL C00703
MOVL C00704
MOVL C00705
MOVL C00706
MOVL C00707
MOVL C00708
MOVL C00709
MOVL C00710
MOVL C00711
MOVL C00712
MOVL C00713
MOVL C00714
MOVL C00715
MOVL C00716
MOVL C00717
MOVL C00718
MOVL C00719
MOVL C00720
MOVL C00721
MOVL C00722
MOVL C00723
MOVL C00724
MOVL C00725
MOVL C00726
MOVL C00727
MOVL C00728
MOVL C00729
MOVL C00730
MOVL C00731
MOVL C00732
MOVL C00733
MOVL C00734
MOVL C00735
MOVL C00736
MOVL C00737
MOVL C00738
MOVL C00739
MOVL C00740
MOVL C00741
MOVL C00742
MOVL C00743
MOVL C00744
MOVL C00745
MOVL C00746
MOVL C00747
MOVL C00748
MOVL C00749
MOVL C00750
MOVL C00751
MOVL C00752
MOVL C00753
MOVL C00754
MOVL C00755
MOVL C00756
MOVL C00757
MOVL C00758
MOVL C00759
MOVL C00760
MOVL C00761
MOVL C00762
MOVL C00763
MOVL C00764
MOVL C00765
MOVL C00766
MOVL C00767
MOVL C00768
MOVL C00769
MOVL C00770
MOVL C00771
MOVL C00772
MOVL C00773
MOVL C00774
MOVL C00775
MOVL C00776
MOVL C00777
MOVL C00778
MOVL C00779
MOVL C00780
MOVL C00781
MOVL C00782
MOVL C00783
MOVL C00784
MOVL C00785
MOVL C00786
MOVL C00787
MOVL C00788
MOVL C00789
MOVL C00790
MOVL C00791
MOVL C00792
MOVL C00793
MOVL C00794
MOVL C00795
MOVL C00796
MOVL C00797
MOVL C00798
MOVL C00799
MOVL C00800
MOVL C00801
MOVL C00802
MOVL C00803
MOVL C00804
MOVL C00805
MOVL C00806
MOVL C00807
MOVL C00808
MOVL C00809
MOVL C00810
MOVL C00811
MOVL C00812
MOVL C00813
MOVL C00814
MOVL C00815
MOVL C00816
MOVL C00817
MOVL C00818
MOVL C00819
MOVL C00820
MOVL C00821
MOVL C00822
MOVL C00823
MOVL C00824
MOVL C00825
MOVL C00826
MOVL C00827
MOVL C00828
MOVL C00829
MOVL C00830
MOVL C00831
MOVL C00832
MOVL C00833
MOVL C00834
MOVL C00835
MOVL C00836
MOVL C00837
MOVL C00838
MOVL C00839
MOVL C00840
MOVL C00841
MOVL C00842
MOVL C00843
MOVL C00844
MOVL C00845
MOVL C00846
MOVL C00847
MOVL C00848
MOVL C00849
MOVL C00850
MOVL C00851
MOVL C00852
MOVL C00853
MOVL C00854
MOVL C00855
MOVL C00856
MOVL C00857
MOVL C00858
MOVL C00859
MOVL C00860
MOVL C00861
MOVL C00862
MOVL C00863
MOVL C00864
MOVL C00865
MOVL C00866
MOVL C00867
MOVL C00868
MOVL C00869
MOVL C00870
MOVL C00871
MOVL C00872
MOVL C00873
MOVL C00874
MOVL C00875
MOVL C00876
MOVL C00877
MOVL C00878
MOVL C00879
MOVL C00880
MOVL C00881
MOVL C00882
MOVL C00883
MOVL C00884
MOVL C00885
MOVL C00886
MOVL C00887
MOVL C00888
MOVL C00889
MOVL C00890
MOVL C00891
MOVL C00892
MOVL C00893
MOVL C00894
MOVL C00895
MOVL C00896
MOVL C00897
ARCOF
MOVL C00898
ARCON
MOVL C00899
MOVL C00900
MOVL C00901
MOVL C00902
MOVL C00903
MOVL C00904
MOVL C00905
MOVL C00906
MOVL C00907
MOVL C00908
MOVL C00909
MOVL C00910
MOVL C00911
MOVL C00912
MOVL C00913
MOVL C00914
MOVL C00915
MOVL C00916
ARCOF
MOVL C00917
ARCON
MOVL C00918
MOVL C00919
MOVL C00920
MOVL C00921
MOVL C00922
MOVL C00923
MOVL C00924
MOVL C00925
MOVL C00926
MOVL C00927
MOVL C00928
MOVL C00929
MOVL C00930
MOVL C00931
MOVL C00932
MOVL C00933
MOVL C00934
MOVL C00935
ARCOF
MOVL C00936
ARCON
MOVL C00937
MOVL C00938
MOVL C00939
MOVL C00940
MOVL C00941
MOVL C00942
MOVL C00943
MOVL C00944
MOVL C00945
MOVL C00946
MOVL C00947
MOVL C00948
MOVL C00949
MOVL C00950
MOVL C00951
MOVL C00952
MOVL C00953
MOVL C00954
ARCOF
MOVL C00955
ARCON
MOVL C00956
MOVL C00957
MOVL C00958
MOVL C00959
MOVL C00960
MOVL C00961
MOVL C00962
MOVL C00963
MOVL C00964
MOVL C00965
MOVL C00966
MOVL C00967
MOVL C00968
MOVL C00969
MOVL C00970
MOVL C00971
MOVL C00972
MOVL C00973
MOVL C00974
ARCOF
MOVL C00975
ARCON
MOVL C00976
MOVL C00977
MOVL C00978
MOVL C00979
MOVL C00980
MOVL C00981
MOVL C00982
MOVL C00983
MOVL C00984
MOVL C00985
MOVL C00986
MOVL C00987
MOVL C00988
MOVL C00989
MOVL C00990
MOVL C00991
MOVL C00992
MOVL C00993
ARCOF
MOVL C00994
ARCON
MOVL C00995
MOVL C00996
MOVL C00997
MOVL C00998
MOVL C00999
MOVL C01000
MOVL C01001
MOVL C01002
MOVL C01003
MOVL C01004
MOVL C01005
MOVL C01006
MOVL C01007
MOVL C01008
MOVL C01009
MOVL C01010
MOVL C01011
MOVL C01012
ARCOF
MOVL C01013
ARCON
MOVL C01014
MOVL C01015
MOVL C01016
MOVL C01017
MOVL C01018
MOVL C01019
MOVL C01020
MOVL C01021
MOVL C01022
MOVL C01023
MOVL C01024
MOVL C01025
MOVL C01026
MOVL C01027
MOVL C01028
MOVL C01029
MOVL C01030
MOVL C01031
ARCOF
MOVL C01032
ARCON
MOVL C01033
MOVL C01034
MOVL C01035
MOVL C01036
MOVL C01037
MOVL C01038
MOVL C01039
MOVL C01040
MOVL C01041
MOVL C01042
MOVL C01043
MOVL C01044
MOVL C01045
MOVL C01046
MOVL C01047
MOVL C01048
ARCOF
MOVL C01049
ARCON
MOVL C01050
MOVL C01051
MOVL C01052
MOVL C01053
MOVL C01054
MOVL C01055
MOVL C01056
MOVL C01057
MOVL C01058
MOVL C01059
MOVL C01060
MOVL C01061
ARCOF
MOVL C01062
ARCON
MOVL C01063
MOVL C01064
MOVL C01065
MOVL C01066
MOVL C01067
MOVL C01068
MOVL C01069
MOVL C01070
MOVL C01071
MOVL C01072
MOVL C01073
MOVL C01074
ARCOF
MOVL C01075
ARCON
MOVL C01076
MOVL C01077
MOVL C01078
MOVL C01079
MOVL C01080
MOVL C01081
MOVL C01082
MOVL C01083
MOVL C01084
MOVL C01085
MOVL C01086
MOVL C01087
ARCOF
MOVL C01088
ARCON
MOVL C01089
MOVL C01090
MOVL C01091
MOVL C01092
MOVL C01093
MOVL C01094
MOVL C01095
MOVL C01096
MOVL C01097
MOVL C01098
MOVL C01099
MOVL C01100
MOVL C01101
ARCOF
MOVL C01102
ARCON
MOVL C01103
MOVL C01104
MOVL C01105
MOVL C01106
MOVL C01107
MOVL C01108
MOVL C01109
MOVL C01110
MOVL C01111
MOVL C01112
MOVL C01113
MOVL C01114
ARCOF
MOVL C01115
ARCON
MOVL C01116
MOVL C01117
MOVL C01118
MOVL C01119
MOVL C01120
MOVL C01121
MOVL C01122
MOVL C01123
MOVL C01124
MOVL C01125
MOVL C01126
MOVL C01127
ARCOF
MOVL C01128
ARCON
MOVL C01129
MOVL C01130
MOVL C01131
MOVL C01132
MOVL C01133
MOVL C01134
MOVL C01135
MOVL C01136
MOVL C01137
MOVL C01138
MOVL C01139
MOVL C01140
ARCOF
MOVL C01141
ARCON
MOVL C01142
MOVL C01143
MOVL C01144
MOVL C01145
MOVL C01146
MOVL C01147
MOVL C01148
MOVL C01149
MOVL C01150
MOVL C01151
MOVL C01152
MOVL C01153
ARCOF
MOVL C01154
ARCON
MOVL C01155
MOVL C01156
MOVL C01157
MOVL C01158
MOVL C01159
MOVL C01160
MOVL C01161
MOVL C01162
MOVL C01163
MOVL C01164
ARCOF
MOVL C01165
ARCON
MOVL C01166
MOVL C01167
MOVL C01168
MOVL C01169
MOVL C01170
MOVL C01171
MOVL C01172
MOVL C01173
MOVL C01174
MOVL C01175
ARCOF
MOVL C01176
ARCON
MOVL C01177
MOVL C01178
MOVL C01179
MOVL C01180
MOVL C01181
MOVL C01182
MOVL C01183
MOVL C01184
MOVL C01185
MOVL C01186
ARCOF
MOVL C01187
ARCON
MOVL C01188
MOVL C01189
MOVL C01190
MOVL C01191
MOVL C01192
MOVL C01193
MOVL C01194
MOVL C01195
MOVL C01196
MOVL C01197
MOVL C01198
ARCOF
MOVL C01199
ARCON
MOVL C01200
MOVL C01201
MOVL C01202
MOVL C01203
MOVL C01204
MOVL C01205
MOVL C01206
MOVL C01207
MOVL C01208
MOVL C01209
ARCOF
MOVL C01210
ARCON
MOVL C01211
MOVL C01212
MOVL C01213
MOVL C01214
MOVL C01215
MOVL C01216
MOVL C01217
MOVL C01218
MOVL C01219
MOVL C01220
ARCOF
MOVL C01221
ARCON
MOVL C01222
MOVL C01223
MOVL C01224
MOVL C01225
MOVL C01226
MOVL C01227
MOVL C01228
MOVL C01229
MOVL C01230
MOVL C01231
ARCOF
MOVL C01232
ARCON
MOVL C01233
MOVL C01234
MOVL C01235
MOVL C01236
MOVL C01237
MOVL C01238
MOVL C01239
MOVL C01240
MOVL C01241
MOVL C01242
MOVL C01243
ARCOF
MOVL C01244
ARCON
MOVL C01245
MOVL C01246
MOVL C01247
MOVL C01248
MOVL C01249
MOVL C01250
MOVL C01251
MOVL C01252
MOVL C01253
MOVL C01254
ARCOF
MOVL C01255
ARCON
MOVL C01256
MOVL C01257
MOVL C01258
MOVL C01259
MOVL C01260
MOVL C01261
MOVL C01262
MOVL C01263
MOVL C01264
MOVL C01265
ARCOF
MOVL C01266
ARCON
MOVL C01267
MOVL C01268
MOVL C01269
MOVL C01270
MOVL C01271
MOVL C01272
MOVL C01273
MOVL C01274
MOVL C01275
MOVL C01276
ARCOF
MOVL C01277
ARCON
MOVL C01278
MOVL C01279
MOVL C01280
MOVL C01281
MOVL C01282
MOVL C01283
MOVL C01284
MOVL C01285
MOVL C01286
MOVL C01287
MOVL C01288
ARCOF
MOVL C01289
ARCON
MOVL C01290
MOVL C01291
MOVL C01292
MOVL C01293
MOVL C01294
MOVL C01295
MOVL C01296
MOVL C01297
MOVL C01298
MOVL C01299
ARCOF
MOVL C01300
ARCON
MOVL C01301
MOVL C01302
MOVL C01303
MOVL C01304
MOVL C01305
MOVL C01306
MOVL C01307
MOVL C01308
MOVL C01309
MOVL C01310
ARCOF
MOVL C01311
ARCON
MOVL C01312
MOVL C01313
MOVL C01314
MOVL C01315
MOVL C01316
MOVL C01317
MOVL C01318
MOVL C01319
MOVL C01320
MOVL C01321
ARCOF
MOVL C01322
ARCON
MOVL C01323
MOVL C01324
MOVL C01325
MOVL C01326
MOVL C01327
MOVL C01328
MOVL C01329
MOVL C01330
MOVL C01331
MOVL C01332
ARCOF
MOVL C01333
ARCON
MOVL C01334
MOVL C01335
MOVL C01336
MOVL C01337
MOVL C01338
MOVL C01339
MOVL C01340
MOVL C01341
ARCOF
MOVL C01342
ARCON
MOVL C01343
MOVL C01344
MOVL C01345
MOVL C01346
MOVL C01347
MOVL C01348
MOVL C01349
MOVL C01350
ARCOF
MOVL C01351
ARCON
MOVL C01352
MOVL C01353
MOVL C01354
MOVL C01355
MOVL C01356
MOVL C01357
MOVL C01358
MOVL C01359
ARCOF
MOVL C01360
ARCON
MOVL C01361
MOVL C01362
MOVL C01363
MOVL C01364
MOVL C01365
MOVL C01366
MOVL C01367
MOVL C01368
MOVL C01369
ARCOF
MOVL C01370
ARCON
MOVL C01371
MOVL C01372
MOVL C01373
MOVL C01374
MOVL C01375
MOVL C01376
MOVL C01377
MOVL C01378
ARCOF
MOVL C01379
ARCON
MOVL C01380
MOVL C01381
MOVL C01382
MOVL C01383
MOVL C01384
MOVL C01385
MOVL C01386
MOVL C01387
ARCOF
MOVL C01388
ARCON
MOVL C01389
MOVL C01390
MOVL C01391
MOVL C01392
MOVL C01393
MOVL C01394
MOVL C01395
MOVL C01396
ARCOF
MOVL C01397
ARCON
MOVL C01398
MOVL C01399
MOVL C01400
MOVL C01401
MOVL C01402
MOVL C01403
MOVL C01404
MOVL C01405
ARCOF
MOVL C01406
ARCON
MOVL C01407
MOVL C01408
MOVL C01409
MOVL C01410
MOVL C01411
MOVL C01412
ARCOF
MOVL C01413
ARCON
MOVL C01414
MOVL C01415
MOVL C01416
MOVL C01417
MOVL C01418
MOVL C01419
ARCOF
MOVL C01420
ARCON
MOVL C01421
MOVL C01422
MOVL C01423
MOVL C01424
MOVL C01425
MOVL C01426
ARCOF
MOVL C01427
ARCON
MOVL C01428
MOVL C01429
MOVL C01430
MOVL C01431
MOVL C01432
MOVL C01433
MOVL C01434
ARCOF
MOVL C01435
ARCON
MOVL C01436
MOVL C01437
MOVL C01438
MOVL C01439
MOVL C01440
MOVL C01441
ARCOF
MOVL C01442
ARCON
MOVL C01443
MOVL C01444
MOVL C01445
MOVL C01446
MOVL C01447
MOVL C01448
ARCOF
MOVL C01449
ARCON
MOVL C01450
MOVL C01451
MOVL C01452
MOVL C01453
MOVL C01454
MOVL C01455
ARCOF
MOVL C01456
ARCON
MOVL C01457
MOVL C01458
MOVL C01459
MOVL C01460
MOVL C01461
MOVL C01462
MOVL C01463
ARCOF
MOVL C01464
ARCON
MOVL C01465
MOVL C01466
MOVL C01467
MOVL C01468
MOVL C01469
MOVL C01470
ARCOF
MOVL C01471
ARCON
MOVL C01472
MOVL C01473
MOVL C01474
MOVL C01475
MOVL C01476
MOVL C01477
ARCOF
MOVL C01478
ARCON
MOVL C01479
MOVL C01480
MOVL C01481
MOVL C01482
MOVL C01483
MOVL C01484
ARCOF
MOVL C01485
ARCON
MOVL C01486
MOVL C01487
MOVL C01488
MOVL C01489
MOVL C01490
MOVL C01491
MOVL C01492
ARCOF
MOVL C01493
ARCON
MOVL C01494
MOVL C01495
MOVL C01496
MOVL C01497
MOVL C01498
MOVL C01499
ARCOF
MOVL C01500
ARCON
MOVL C01501
MOVL C01502
MOVL C01503
MOVL C01504
MOVL C01505
MOVL C01506
ARCOF
MOVL C01507
ARCON
MOVL C01508
MOVL C01509
MOVL C01510
MOVL C01511
MOVL C01512
MOVL C01513
ARCOF
MOVL C01514
ARCON
MOVL C01515
MOVL C01516
MOVL C01517
END
